   LIN {X -9.091, Y -16.998, Z 51.850} C_DIS
   LIN {X -7.957, Y -14.503, Z 51.850} C_DIS
   LIN {X -6.497, Y -10.839, Z 51.850} C_DIS
   LIN {X -6.440, Y -10.684, Z 51.850} C_DIS
   LIN {X -5.101, Y -6.672, Z 51.850} C_DIS
   LIN {X -4.128, Y -3.010, Z 51.850} C_DIS
   LIN {X -3.893, Y -2.128, Z 51.850} C_DIS
   LIN {X -3.542, Y -0.234, Z 51.850} C_DIS
   LIN {X -2.837, Y 3.485, Z 51.850} C_DIS
   LIN {X -2.656, Y 4.674, Z 51.850} C_DIS
   LIN {X -2.279, Y 9.653, Z 51.850} C_DIS
   LIN {X -2.115, Y 11.765, Z 51.850} C_DIS
   LIN {X -2.086, Y 12.130, Z 51.850} C_DIS
   LIN {X -2.030, Y 12.659, Z 51.850} C_DIS
   LIN {X -2.082, Y 13.927, Z 51.850} C_DIS
   LIN {X -2.664, Y 23.969, Z 51.850} C_DIS
   LIN {X -2.957, Y 25.919, Z 51.850} C_DIS
   LIN {X -3.415, Y 28.463, Z 51.850} C_DIS
   LIN {X -3.462, Y 28.724, Z 51.850} C_DIS
   LIN {X -3.657, Y 29.589, Z 51.850} C_DIS
   LIN {X -4.174, Y 31.893, Z 51.850} C_DIS
   LIN {X -4.435, Y 32.885, Z 51.850} C_DIS
   LIN {X -4.782, Y 34.185, Z 51.850} C_DIS
   LIN {X -5.293, Y 35.880, Z 51.850} C_DIS
   LIN {X -5.465, Y 36.456, Z 51.850} C_DIS
   LIN {X -5.565, Y 36.761, Z 51.850} C_DIS
   LIN {X -5.967, Y 37.975, Z 51.850} C_DIS
   LIN {X -6.308, Y 38.961, Z 51.850} C_DIS
   LIN {X -6.377, Y 39.157, Z 51.850} C_DIS
   LIN {X -6.424, Y 39.407, Z 51.850} C_DIS
   LIN {X -6.622, Y 40.453, Z 51.850} C_DIS
   LIN {X -6.434, Y 41.604, Z 51.850} C_DIS
   LIN {X -6.389, Y 41.872, Z 51.850} C_DIS
   LIN {X -6.240, Y 42.112, Z 51.850} C_DIS
   LIN {X -5.463, Y 43.327, Z 51.850} C_DIS
   LIN {X -3.784, Y 44.088, Z 51.850} C_DIS
   LIN {X -2.954, Y 44.485, Z 51.850} C_DIS
   LIN {X -2.346, Y 44.397, Z 51.850} C_DIS
   LIN {X -1.227, Y 44.232, Z 51.850}
   LaserEnd_Ext()
   LIN {X 8.602, Y 5.790, Z 51.850}
   LaserStart_Ext()
   LIN {X 8.602, Y -9.042, Z 51.850}
   LaserEnd_Ext()
   LIN {X 7.602, Y -17.948, Z 51.850}
   LaserStart_Ext()
   LIN {X 7.602, Y 15.368, Z 51.850}
   LaserEnd_Ext()
   LIN {X 6.602, Y 20.531, Z 51.850}
   LaserStart_Ext()
   LIN {X 6.602, Y -22.967, Z 51.850}
   LaserEnd_Ext()
   LIN {X 5.602, Y -25.282, Z 51.850}
   LaserStart_Ext()
   LIN {X 5.602, Y 25.306, Z 51.850}
   LaserEnd_Ext()
   LIN {X 4.602, Y 28.856, Z 51.850}
   LaserStart_Ext()
   LIN {X 4.602, Y -19.113, Z 51.850}
   LaserEnd_Ext()
   LIN {X 4.602, Y -22.901, Z 51.850}
   LaserStart_Ext()
   LIN {X 4.602, Y -26.434, Z 51.850}
   LaserEnd_Ext()
   LIN {X 3.602, Y -27.404, Z 51.850}
   LaserStart_Ext()
   LIN {X 3.602, Y -24.729, Z 51.850}
   LaserEnd_Ext()
   LIN {X 3.602, Y -17.421, Z 51.850}
   LaserStart_Ext()
   LIN {X 3.602, Y 32.251, Z 51.850}
   LaserEnd_Ext()
   LIN {X 2.602, Y 35.260, Z 51.850}
   LaserStart_Ext()
   LIN {X 2.602, Y -16.373, Z 51.850}
   LaserEnd_Ext()
   LIN {X 2.602, Y -25.693, Z 51.850}
   LaserStart_Ext()
   LIN {X 2.602, Y -27.986, Z 51.850}
   LaserEnd_Ext()
   LIN {X 1.602, Y -28.384, Z 51.850}
   LaserStart_Ext()
   LIN {X 1.602, Y -26.285, Z 51.850}
   LaserEnd_Ext()
   LIN {X 1.602, Y -15.740, Z 51.850}
   LaserStart_Ext()
   LIN {X 1.602, Y 37.974, Z 51.850}
   LaserEnd_Ext()
   LIN {X 0.602, Y 40.498, Z 51.850}
   LaserStart_Ext()
   LIN {X 0.602, Y -15.317, Z 51.850}
   LaserEnd_Ext()
   LIN {X 0.602, Y -26.624, Z 51.850}
   LaserStart_Ext()
   LIN {X 0.602, Y -28.775, Z 51.850}
   LaserEnd_Ext()
   LIN {X -0.398, Y -28.815, Z 51.850}
   LaserStart_Ext()
   LIN {X -0.398, Y -26.985, Z 51.850}
   LaserEnd_Ext()
   LIN {X -0.398, Y -15.189, Z 51.850}
   LaserStart_Ext()
   LIN {X -0.398, Y 42.404, Z 51.850}
   LaserEnd_Ext()
   LIN {X -1.398, Y 43.147, Z 51.850}
   LaserStart_Ext()
   LIN {X -1.398, Y 19.405, Z 51.850}
   LaserEnd_Ext()
   LIN {X -1.398, Y 8.047, Z 51.850}
   LaserStart_Ext()
   LIN {X -1.398, Y -15.067, Z 51.850}
   LaserEnd_Ext()
   LIN {X -1.398, Y -26.955, Z 51.850}
   LaserStart_Ext()
   LIN {X -1.398, Y -28.642, Z 51.850}
   LaserEnd_Ext()
   LIN {X -2.398, Y -28.469, Z 51.850}
   LaserStart_Ext()
   LIN {X -2.398, Y -26.818, Z 51.850}
   LaserEnd_Ext()
   LIN {X -2.398, Y -15.309, Z 51.850}
   LaserStart_Ext()
   LIN {X -2.398, Y 0.432, Z 51.850}
   LaserEnd_Ext()
   LIN {X -2.398, Y 28.460, Z 51.850}
   LaserStart_Ext()
   LIN {X -2.398, Y 43.394, Z 51.850}
   LaserEnd_Ext()
   LIN {X -3.398, Y 43.165, Z 51.850}
   LaserStart_Ext()
   LIN {X -3.398, Y 32.873, Z 51.850}
   LaserEnd_Ext()
   LIN {X -3.398, Y -4.158, Z 51.850}
   LaserStart_Ext()
   LIN {X -3.398, Y -15.630, Z 51.850}
   LaserEnd_Ext()
   LIN {X -3.398, Y -26.558, Z 51.850}
   LaserStart_Ext()
   LIN {X -3.398, Y -28.295, Z 51.850}
   LaserEnd_Ext()
   LIN {X -4.398, Y -28.122, Z 51.850}
   LaserStart_Ext()
   LIN {X -4.398, Y -25.932, Z 51.850}
   LaserEnd_Ext()
   LIN {X -4.398, Y -16.131, Z 51.850}
   LaserStart_Ext()
   LIN {X -4.398, Y -7.724, Z 51.850}
   LaserEnd_Ext()
   LIN {X -4.398, Y 36.378, Z 51.850}
   LaserStart_Ext()
   LIN {X -4.398, Y 42.712, Z 51.850}
   LaserEnd_Ext()
   LIN {X -5.398, Y 41.572, Z 51.850}
   LaserStart_Ext()
   LIN {X -5.398, Y 39.387, Z 51.850}
   LaserEnd_Ext()
   LIN {X -5.398, Y -10.720, Z 51.850}
   LaserStart_Ext()
   LIN {X -5.398, Y -17.051, Z 51.850}
   LaserEnd_Ext()
   LIN {X -5.398, Y -25.183, Z 51.850}
   LaserStart_Ext()
   LIN {X -5.398, Y -27.718, Z 51.850}
   LaserEnd_Ext()
   LIN {X -6.398, Y -26.934, Z 51.850}
   LaserStart_Ext()
   LIN {X -6.398, Y -23.699, Z 51.850}
   LaserEnd_Ext()
   LIN {X -6.398, Y -18.786, Z 51.850}
   LaserStart_Ext()
   LIN {X -6.398, Y -13.293, Z 51.850}
   LaserEnd_Ext()
   LIN {X -7.398, Y -15.691, Z 51.850}
   LaserStart_Ext()
   LIN {X -7.398, Y -25.741, Z 51.850}
   LaserEnd_Ext()
   LIN {X -8.398, Y -24.042, Z 51.850}
   LaserStart_Ext()
   LIN {X -8.398, Y -18.107, Z 51.850}
   LaserEnd_Ext()
   LIN {X 3.897, Y -22.048, Z 52.700}
   LaserStart_Ext()
   LIN {X 3.461, Y -23.044, Z 52.700} C_DIS
   LIN {X 3.108, Y -23.846, Z 52.700} C_DIS
   LIN {X 1.957, Y -24.884, Z 52.700} C_DIS
   LIN {X 1.508, Y -25.317, Z 52.700} C_DIS
   LIN {X 0.879, Y -25.530, Z 52.700} C_DIS
   LIN {X -0.660, Y -25.986, Z 52.700} C_DIS
   LIN {X -1.668, Y -25.850, Z 52.700} C_DIS
   LIN {X -2.710, Y -25.707, Z 52.700} C_DIS
   LIN {X -3.925, Y -24.947, Z 52.700} C_DIS
   LIN {X -4.462, Y -24.613, Z 52.700} C_DIS
   LIN {X -4.766, Y -24.167, Z 52.700} C_DIS
   LIN {X -5.630, Y -22.888, Z 52.700} C_DIS
   LIN {X -5.881, Y -21.409, Z 52.700} C_DIS
   LIN {X -5.980, Y -20.831, Z 52.700} C_DIS
   LIN {X -5.800, Y -20.305, Z 52.700} C_DIS
   LIN {X -5.042, Y -18.100, Z 52.700} C_DIS
   LIN {X -3.563, Y -16.747, Z 52.700} C_DIS
   LIN {X -3.489, Y -16.679, Z 52.700} C_DIS
   LIN {X -1.401, Y -16.013, Z 52.700} C_DIS
   LIN {X 0.253, Y -16.220, Z 52.700} C_DIS
   LIN {X 0.741, Y -16.280, Z 52.700} C_DIS
   LIN {X 1.229, Y -16.586, Z 52.700} C_DIS
   LIN {X 2.539, Y -17.413, Z 52.700} C_DIS
   LIN {X 3.482, Y -19.002, Z 52.700} C_DIS
   LIN {X 3.839, Y -19.599, Z 52.700} C_DIS
   LIN {X 3.868, Y -20.120, Z 52.700} C_DIS
   LIN {X 3.897, Y -22.048, Z 52.700}
   LaserEnd_Ext()
   LIN {X -6.440, Y 39.195, Z 52.700}
   LaserStart_Ext()
   LIN {X -6.031, Y 38.023, Z 52.700} C_DIS
   LIN {X -5.522, Y 36.495, Z 52.700} C_DIS
   LIN {X -5.003, Y 34.786, Z 52.700} C_DIS
   LIN {X -4.834, Y 34.226, Z 52.700} C_DIS
   LIN {X -4.622, Y 33.433, Z 52.700} C_DIS
   LIN {X -4.220, Y 31.936, Z 52.700} C_DIS
   LIN {X -4.160, Y 31.686, Z 52.700} C_DIS
   LIN {X -3.517, Y 28.844, Z 52.700} C_DIS
   LIN {X -3.238, Y 27.287, Z 52.700} C_DIS
   LIN {X -2.907, Y 25.444, Z 52.700} C_DIS
   LIN {X -2.694, Y 24.032, Z 52.700} C_DIS
   LIN {X -2.042, Y 12.765, Z 52.700} C_DIS
   LIN {X -2.035, Y 12.665, Z 52.700} C_DIS
   LIN {X -2.630, Y 4.802, Z 52.700} C_DIS
   LIN {X -2.918, Y 2.908, Z 52.700} C_DIS
   LIN {X -3.872, Y -2.129, Z 52.700} C_DIS
   LIN {X -3.961, Y -2.483, Z 52.700} C_DIS
   LIN {X -4.159, Y -3.222, Z 52.700} C_DIS
   LIN {X -5.120, Y -6.839, Z 52.700} C_DIS
   LIN {X -5.819, Y -8.933, Z 52.700} C_DIS
   LIN {X -6.431, Y -10.775, Z 52.700} C_DIS
   LIN {X -7.191, Y -12.703, Z 52.700} C_DIS
   LIN {X -7.896, Y -14.470, Z 52.700} C_DIS
   LIN {X -8.539, Y -15.886, Z 52.700} C_DIS
   LIN {X -9.111, Y -17.160, Z 52.700} C_DIS
   LIN {X -9.455, Y -18.416, Z 52.700} C_DIS
   LIN {X -9.956, Y -20.216, Z 52.700} C_DIS
   LIN {X -9.683, Y -22.635, Z 52.700} C_DIS
   LIN {X -9.534, Y -23.902, Z 52.700} C_DIS
   LIN {X -8.671, Y -25.359, Z 52.700} C_DIS
   LIN {X -7.628, Y -27.131, Z 52.700} C_DIS
   LIN {X -6.992, Y -27.631, Z 52.700} C_DIS
   LIN {X -5.335, Y -28.917, Z 52.700} C_DIS
   LIN {X -2.287, Y -29.446, Z 52.700} C_DIS
   LIN {X 0.367, Y -29.899, Z 52.700} C_DIS
   LIN {X 2.301, Y -29.198, Z 52.700} C_DIS
   LIN {X 3.776, Y -28.611, Z 52.700} C_DIS
   LIN {X 4.726, Y -27.690, Z 52.700} C_DIS
   LIN {X 6.373, Y -26.159, Z 52.700} C_DIS
   LIN {X 7.607, Y -23.279, Z 52.700} C_DIS
   LIN {X 7.870, Y -22.673, Z 52.700} C_DIS
   LIN {X 7.953, Y -22.225, Z 52.700} C_DIS
   LIN {X 8.447, Y -19.461, Z 52.700} C_DIS
   LIN {X 8.873, Y -16.648, Z 52.700} C_DIS
   LIN {X 8.891, Y -16.534, Z 52.700} C_DIS
   LIN {X 8.906, Y -16.414, Z 52.700} C_DIS
   LIN {X 9.346, Y -12.755, Z 52.700} C_DIS
   LIN {X 9.568, Y -10.105, Z 52.700} C_DIS
   LIN {X 9.732, Y -7.982, Z 52.700} C_DIS
   LIN {X 9.893, Y -2.443, Z 52.700} C_DIS
   LIN {X 9.924, Y -1.495, Z 52.700} C_DIS
   LIN {X 9.827, Y 1.258, Z 52.700} C_DIS
   LIN {X 9.794, Y 2.098, Z 52.700} C_DIS
   LIN {X 9.781, Y 4.353, Z 52.700} C_DIS
   LIN {X 9.137, Y 10.313, Z 52.700} C_DIS
   LIN {X 8.700, Y 14.833, Z 52.700} C_DIS
   LIN {X 7.579, Y 20.715, Z 52.700} C_DIS
   LIN {X 6.563, Y 25.567, Z 52.700} C_DIS
   LIN {X 5.392, Y 29.673, Z 52.700} C_DIS
   LIN {X 4.526, Y 32.613, Z 52.700} C_DIS
   LIN {X 4.051, Y 34.041, Z 52.700} C_DIS
   LIN {X 3.564, Y 35.455, Z 52.700} C_DIS
   LIN {X 3.153, Y 36.583, Z 52.700} C_DIS
   LIN {X 2.877, Y 37.340, Z 52.700} C_DIS
   LIN {X 2.446, Y 38.454, Z 52.700} C_DIS
   LIN {X 2.118, Y 39.311, Z 52.700} C_DIS
   LIN {X 1.886, Y 39.889, Z 52.700} C_DIS
   LIN {X 1.543, Y 40.733, Z 52.700} C_DIS
   LIN {X 1.075, Y 41.846, Z 52.700} C_DIS
   LIN {X 0.968, Y 42.102, Z 52.700} C_DIS
   LIN {X 0.846, Y 42.287, Z 52.700} C_DIS
   LIN {X 0.152, Y 43.327, Z 52.700} C_DIS
   LIN {X -1.096, Y 44.147, Z 52.700} C_DIS
   LIN {X -1.303, Y 44.282, Z 52.700} C_DIS
   LIN {X -1.744, Y 44.345, Z 52.700} C_DIS
   LIN {X -3.030, Y 44.531, Z 52.700} C_DIS
   LIN {X -5.347, Y 43.424, Z 52.700} C_DIS
   LIN {X -5.565, Y 43.330, Z 52.700} C_DIS
   LIN {X -5.657, Y 43.211, Z 52.700} C_DIS
   LIN {X -6.452, Y 41.928, Z 52.700} C_DIS
   LIN {X -6.652, Y 40.735, Z 52.700} C_DIS
   LIN {X -6.689, Y 40.519, Z 52.700} C_DIS
   LIN {X -6.649, Y 40.300, Z 52.700} C_DIS
   LIN {X -6.440, Y 39.195, Z 52.700}
   LaserEnd_Ext()
   LIN {X -0.513, Y 42.522, Z 52.700}
   LaserStart_Ext()
   LIN {X -4.907, Y 42.522, Z 52.700}
   LaserEnd_Ext()
   LIN {X -5.506, Y 41.522, Z 52.700}
   LaserStart_Ext()
   LIN {X 0.127, Y 41.522, Z 52.700}
   LaserEnd_Ext()
   LIN {X 0.547, Y 40.522, Z 52.700}
   LaserStart_Ext()
   LIN {X -5.673, Y 40.522, Z 52.700}
   LaserEnd_Ext()
   LIN {X -5.484, Y 39.522, Z 52.700}
   LaserStart_Ext()
   LIN {X 0.956, Y 39.522, Z 52.700}
   LaserEnd_Ext()
   LIN {X 1.350, Y 38.522, Z 52.700}
   LaserStart_Ext()
   LIN {X -5.146, Y 38.522, Z 52.700}
   LaserEnd_Ext()
   LIN {X -4.810, Y 37.522, Z 52.700}
   LaserStart_Ext()
   LIN {X 1.735, Y 37.522, Z 52.700}
   LaserEnd_Ext()
   LIN {X 2.111, Y 36.522, Z 52.700}
   LaserStart_Ext()
   LIN {X -4.485, Y 36.522, Z 52.700}
   LaserEnd_Ext()
   LIN {X -4.181, Y 35.522, Z 52.700}
   LaserStart_Ext()
   LIN {X 2.475, Y 35.522, Z 52.700}
   LaserEnd_Ext()
   LIN {X 2.828, Y 34.522, Z 52.700}
   LaserStart_Ext()
   LIN {X -3.879, Y 34.522, Z 52.700}
   LaserEnd_Ext()
   LIN {X -3.611, Y 33.522, Z 52.700}
   LaserStart_Ext()
   LIN {X 3.170, Y 33.522, Z 52.700}
   LaserEnd_Ext()
   LIN {X 3.503, Y 32.522, Z 52.700}
   LaserStart_Ext()
   LIN {X -3.342, Y 32.522, Z 52.700}
   LaserEnd_Ext()
   LIN {X -3.097, Y 31.522, Z 52.700}
   LaserStart_Ext()
   LIN {X 3.805, Y 31.522, Z 52.700}
   LaserEnd_Ext()
   LIN {X 4.100, Y 30.522, Z 52.700}
   LaserStart_Ext()
   LIN {X -2.871, Y 30.522, Z 52.700}
   LaserEnd_Ext()
   LIN {X -2.645, Y 29.522, Z 52.700}
   LaserStart_Ext()
   LIN {X 4.394, Y 29.522, Z 52.700}
   LaserEnd_Ext()
   LIN {X 4.681, Y 28.522, Z 52.700}
   LaserStart_Ext()
   LIN {X -2.443, Y 28.522, Z 52.700}
   LaserEnd_Ext()
   LIN {X -2.264, Y 27.522, Z 52.700}
   LaserStart_Ext()
   LIN {X 4.966, Y 27.522, Z 52.700}
   LaserEnd_Ext()
   LIN {X 5.251, Y 26.522, Z 52.700}
   LaserStart_Ext()
   LIN {X -2.084, Y 26.522, Z 52.700}
   LaserEnd_Ext()
   LIN {X -1.907, Y 25.522, Z 52.700}
   LaserStart_Ext()
   LIN {X 5.536, Y 25.522, Z 52.700}
   LaserEnd_Ext()
   LIN {X 5.760, Y 24.522, Z 52.700}
   LaserStart_Ext()
   LIN {X -1.757, Y 24.522, Z 52.700}
   LaserEnd_Ext()
   LIN {X -1.663, Y 23.522, Z 52.700}
   LaserStart_Ext()
   LIN {X 5.969, Y 23.522, Z 52.700}
   LaserEnd_Ext()
   LIN {X 6.179, Y 22.522, Z 52.700}
   LaserStart_Ext()
   LIN {X -1.605, Y 22.522, Z 52.700}
   LaserEnd_Ext()
   LIN {X -1.547, Y 21.522, Z 52.700}
   LaserStart_Ext()
   LIN {X 6.388, Y 21.522, Z 52.700}
   LaserEnd_Ext()
   LIN {X 6.598, Y 20.522, Z 52.700}
   LaserStart_Ext()
   LIN {X -1.489, Y 20.522, Z 52.700}
   LaserEnd_Ext()
   LIN {X -1.431, Y 19.522, Z 52.700}
   LaserStart_Ext()
   LIN {X 6.788, Y 19.522, Z 52.700}
   LaserEnd_Ext()
   LIN {X 6.979, Y 18.522, Z 52.700}
   LaserStart_Ext()
   LIN {X -1.373, Y 18.522, Z 52.700}
   LaserEnd_Ext()
   LIN {X -1.316, Y 17.522, Z 52.700}
   LaserStart_Ext()
   LIN {X 7.169, Y 17.522, Z 52.700}
   LaserEnd_Ext()
   LIN {X 7.360, Y 16.522, Z 52.700}
   LaserStart_Ext()
   LIN {X -1.258, Y 16.522, Z 52.700}
   LaserEnd_Ext()
   LIN {X -1.200, Y 15.522, Z 52.700}
   LaserStart_Ext()
   LIN {X 7.550, Y 15.522, Z 52.700}
   LaserEnd_Ext()
   LIN {X 7.725, Y 14.522, Z 52.700}
   LaserStart_Ext()
   LIN {X -1.142, Y 14.522, Z 52.700}
   LaserEnd_Ext()
   LIN {X -1.084, Y 13.522, Z 52.700}
   LaserStart_Ext()
   LIN {X 7.822, Y 13.522, Z 52.700}
   LaserEnd_Ext()
   LIN {X 7.919, Y 12.522, Z 52.700}
   LaserStart_Ext()
   LIN {X -1.042, Y 12.522, Z 52.700}
   LaserEnd_Ext()
   LIN {X -1.118, Y 11.522, Z 52.700}
   LaserStart_Ext()
   LIN {X 8.015, Y 11.522, Z 52.700}
   LaserEnd_Ext()
   LIN {X 8.112, Y 10.522, Z 52.700}
   LaserStart_Ext()
   LIN {X -1.194, Y 10.522, Z 52.700}
   LaserEnd_Ext()
   LIN {X -1.269, Y 9.522, Z 52.700}
   LaserStart_Ext()
   LIN {X 8.216, Y 9.522, Z 52.700}
   LaserEnd_Ext()
   LIN {X 8.324, Y 8.522, Z 52.700}
   LaserStart_Ext()
   LIN {X -1.345, Y 8.522, Z 52.700}
   LaserEnd_Ext()
   LIN {X -1.421, Y 7.522, Z 52.700}
   LaserStart_Ext()
   LIN {X 8.433, Y 7.522, Z 52.700}
   LaserEnd_Ext()
   LIN {X 8.541, Y 6.522, Z 52.700}
   LaserStart_Ext()
   LIN {X -1.497, Y 6.522, Z 52.700}
   LaserEnd_Ext()
   LIN {X -1.572, Y 5.522, Z 52.700}
   LaserStart_Ext()
   LIN {X 8.649, Y 5.522, Z 52.700}
   LaserEnd_Ext()
   LIN {X 8.757, Y 4.522, Z 52.700}
   LaserStart_Ext()
   LIN {X -1.661, Y 4.522, Z 52.700}
   LaserEnd_Ext()
   LIN {X -1.813, Y 3.522, Z 52.700}
   LaserStart_Ext()
   LIN {X 8.786, Y 3.522, Z 52.700}
   LaserEnd_Ext()
   LIN {X 8.791, Y 2.522, Z 52.700}
   LaserStart_Ext()
   LIN {X -1.974, Y 2.522, Z 52.700}
   LaserEnd_Ext()
   LIN {X -2.163, Y 1.522, Z 52.700}
   LaserStart_Ext()
   LIN {X 8.816, Y 1.522, Z 52.700}
   LaserEnd_Ext()
   LIN {X 8.852, Y 0.522, Z 52.700}
   LaserStart_Ext()
   LIN {X -2.352, Y 0.522, Z 52.700}
   LaserEnd_Ext()
   LIN {X -2.542, Y -0.478, Z 52.700}
   LaserStart_Ext()
   LIN {X 8.888, Y -0.478, Z 52.700}
   LaserEnd_Ext()
   LIN {X 8.923, Y -1.478, Z 52.700}
   LaserStart_Ext()
   LIN {X -2.731, Y -1.478, Z 52.700}
   LaserEnd_Ext()
   LIN {X -2.929, Y -2.478, Z 52.700}
   LaserStart_Ext()
   LIN {X 8.891, Y -2.478, Z 52.700}
   LaserEnd_Ext()
   LIN {X 8.862, Y -3.478, Z 52.700}
   LaserStart_Ext()
   LIN {X -3.192, Y -3.478, Z 52.700}
   LaserEnd_Ext()
   LIN {X -3.458, Y -4.478, Z 52.700}
   LaserStart_Ext()
   LIN {X 8.833, Y -4.478, Z 52.700}
   LaserEnd_Ext()
   LIN {X 8.804, Y -5.478, Z 52.700}
   LaserStart_Ext()
   LIN {X -3.724, Y -5.478, Z 52.700}
   LaserEnd_Ext()
   LIN {X -3.990, Y -6.478, Z 52.700}
   LaserStart_Ext()
   LIN {X 8.775, Y -6.478, Z 52.700}
   LaserEnd_Ext()
   LIN {X 8.746, Y -7.478, Z 52.700}
   LaserStart_Ext()
   LIN {X -4.279, Y -7.478, Z 52.700}
   LaserEnd_Ext()
   LIN {X -4.613, Y -8.478, Z 52.700}
   LaserStart_Ext()
   LIN {X 8.691, Y -8.478, Z 52.700}
   LaserEnd_Ext()
   LIN {X 8.614, Y -9.478, Z 52.700}
   LaserStart_Ext()
   LIN {X -4.947, Y -9.478, Z 52.700}
   LaserEnd_Ext()
   LIN {X -5.279, Y -10.478, Z 52.700}
   LaserStart_Ext()
   LIN {X 8.533, Y -10.478, Z 52.700}
   LaserEnd_Ext()
   LIN {X 8.449, Y -11.478, Z 52.700}
   LaserStart_Ext()
   LIN {X -5.633, Y -11.478, Z 52.700}
   LaserEnd_Ext()
   LIN {X -6.028, Y -12.478, Z 52.700}
   LaserStart_Ext()
   LIN {X 8.365, Y -12.478, Z 52.700}
   LaserEnd_Ext()
   LIN {X 8.252, Y -13.478, Z 52.700}
   LaserStart_Ext()
   LIN {X -6.424, Y -13.478, Z 52.700}
   LaserEnd_Ext()
   LIN {X -6.822, Y -14.478, Z 52.700}
   LaserStart_Ext()
   LIN {X 8.131, Y -14.478, Z 52.700}
   LaserEnd_Ext()
   LIN {X 8.011, Y -15.478, Z 52.700}
   LaserStart_Ext()
   LIN {X 1.345, Y -15.478, Z 52.700}
   LaserEnd_Ext()
   LIN {X -3.016, Y -15.478, Z 52.700}
   LaserStart_Ext()
   LIN {X -7.255, Y -15.478, Z 52.700}
   LaserEnd_Ext()
   LIN {X -7.709, Y -16.478, Z 52.700}
   LaserStart_Ext()
   LIN {X -4.751, Y -16.478, Z 52.700}
   LaserEnd_Ext()
   LIN {X 2.932, Y -16.478, Z 52.700}
   LaserStart_Ext()
   LIN {X 7.887, Y -16.478, Z 52.700}
   LaserEnd_Ext()
   LIN {X 7.736, Y -17.478, Z 52.700}
   LaserStart_Ext()
   LIN {X 3.740, Y -17.478, Z 52.700}
   LaserEnd_Ext()
   LIN {X -5.824, Y -17.478, Z 52.700}
   LaserStart_Ext()
   LIN {X -8.158, Y -17.478, Z 52.700}
   LaserEnd_Ext()
   LIN {X -8.435, Y -18.478, Z 52.700}
   LaserStart_Ext()
   LIN {X -6.229, Y -18.478, Z 52.700}
   LaserEnd_Ext()
   LIN {X 4.334, Y -18.478, Z 52.700}
   LaserStart_Ext()
   LIN {X 7.585, Y -18.478, Z 52.700}
   LaserEnd_Ext()
   LIN {X 7.428, Y -19.478, Z 52.700}
   LaserStart_Ext()
   LIN {X 4.830, Y -19.478, Z 52.700}
   LaserEnd_Ext()
   LIN {X -6.573, Y -19.478, Z 52.700}
   LaserStart_Ext()
   LIN {X -8.713, Y -19.478, Z 52.700}
   LaserEnd_Ext()
   LIN {X -8.920, Y -20.478, Z 52.700}
   LaserStart_Ext()
   LIN {X -6.916, Y -20.478, Z 52.700}
   LaserEnd_Ext()
   LIN {X 4.873, Y -20.478, Z 52.700}
   LaserStart_Ext()
   LIN {X 7.250, Y -20.478, Z 52.700}
   LaserEnd_Ext()
   LIN {X 7.071, Y -21.478, Z 52.700}
   LaserStart_Ext()
   LIN {X 4.889, Y -21.478, Z 52.700}
   LaserEnd_Ext()
   LIN {X -6.883, Y -21.478, Z 52.700}
   LaserStart_Ext()
   LIN {X -8.808, Y -21.478, Z 52.700}
   LaserEnd_Ext()
   LIN {X -8.695, Y -22.478, Z 52.700}
   LaserStart_Ext()
   LIN {X -6.714, Y -22.478, Z 52.700}
   LaserEnd_Ext()
   LIN {X 4.801, Y -22.478, Z 52.700}
   LaserStart_Ext()
   LIN {X 6.865, Y -22.478, Z 52.700}
   LaserEnd_Ext()
   LIN {X 6.434, Y -23.478, Z 52.700}
   LaserStart_Ext()
   LIN {X 4.362, Y -23.478, Z 52.700}
   LaserEnd_Ext()
   LIN {X -6.438, Y -23.478, Z 52.700}
   LaserStart_Ext()
   LIN {X -8.577, Y -23.478, Z 52.700}
   LaserEnd_Ext()
   LIN {X -8.031, Y -24.478, Z 52.700}
   LaserStart_Ext()
   LIN {X -5.762, Y -24.478, Z 52.700}
   LaserEnd_Ext()
   LIN {X 3.881, Y -24.478, Z 52.700}
   LaserStart_Ext()
   LIN {X 6.006, Y -24.478, Z 52.700}
   LaserEnd_Ext()
   LIN {X 5.577, Y -25.478, Z 52.700}
   LaserStart_Ext()
   LIN {X 2.791, Y -25.478, Z 52.700}
   LaserEnd_Ext()
   LIN {X -4.964, Y -25.478, Z 52.700}
   LaserStart_Ext()
   LIN {X -7.441, Y -25.478, Z 52.700}
   LaserEnd_Ext()
   LIN {X -6.840, Y -26.478, Z 52.700}
   LaserStart_Ext()
   LIN {X -3.363, Y -26.478, Z 52.700}
   LaserEnd_Ext()
   LIN {X 1.195, Y -26.478, Z 52.700}
   LaserStart_Ext()
   LIN {X 4.560, Y -26.478, Z 52.700}
   LaserEnd_Ext()
   LIN {X 3.507, Y -27.478, Z 52.700}
   LaserStart_Ext()
   LIN {X -5.558, Y -27.478, Z 52.700}
   LaserEnd_Ext()
   LIN {X -2.010, Y -28.478, Z 52.700}
   LaserStart_Ext()
   LIN {X 1.352, Y -28.478, Z 52.700}
   LaserEnd_Ext()
   LIN {X -2.322, Y -25.700, Z 53.550}
   LaserStart_Ext()
   LIN {X -2.621, Y -25.660, Z 53.550} C_DIS
   LIN {X -2.815, Y -25.541, Z 53.550} C_DIS
   LIN {X -4.376, Y -24.570, Z 53.550} C_DIS
   LIN {X -5.507, Y -22.909, Z 53.550} C_DIS
   LIN {X -5.560, Y -22.779, Z 53.550} C_DIS
   LIN {X -5.903, Y -20.792, Z 53.550} C_DIS
   LIN {X -5.283, Y -18.984, Z 53.550} C_DIS
   LIN {X -4.960, Y -18.043, Z 53.550} C_DIS
   LIN {X -3.418, Y -16.632, Z 53.550} C_DIS
   LIN {X -1.805, Y -16.113, Z 53.550} C_DIS
   LIN {X -1.333, Y -15.963, Z 53.550} C_DIS
   LIN {X -0.975, Y -16.008, Z 53.550} C_DIS
   LIN {X 0.808, Y -16.225, Z 53.550} C_DIS
   LIN {X 2.587, Y -17.340, Z 53.550} C_DIS
   LIN {X 3.913, Y -19.536, Z 53.550} C_DIS
   LIN {X 4.018, Y -21.420, Z 53.550} C_DIS
   LIN {X 4.024, Y -21.790, Z 53.550} C_DIS
   LIN {X 3.940, Y -21.981, Z 53.550} C_DIS
   LIN {X 3.082, Y -23.933, Z 53.550} C_DIS
   LIN {X 1.954, Y -24.949, Z 53.550} C_DIS
   LIN {X 1.520, Y -25.311, Z 53.550} C_DIS
   LIN {X 0.629, Y -25.576, Z 53.550} C_DIS
   LIN {X -0.583, Y -25.935, Z 53.550} C_DIS
   LIN {X -2.322, Y -25.700, Z 53.550}
   LaserEnd_Ext()
   LIN {X -1.378, Y 44.332, Z 53.550}
   LaserStart_Ext()
   LIN {X -2.427, Y 44.482, Z 53.550} C_DIS
   LIN {X -3.106, Y 44.576, Z 53.550} C_DIS
   LIN {X -3.989, Y 44.311, Z 53.550} C_DIS
   LIN {X -4.992, Y 43.880, Z 53.550} C_DIS
   LIN {X -5.741, Y 43.267, Z 53.550} C_DIS
   LIN {X -6.331, Y 42.297, Z 53.550} C_DIS
   LIN {X -6.511, Y 41.995, Z 53.550} C_DIS
   LIN {X -6.587, Y 41.589, Z 53.550} C_DIS
   LIN {X -6.756, Y 40.620, Z 53.550} C_DIS
   LIN {X -6.582, Y 39.670, Z 53.550} C_DIS
   LIN {X -6.504, Y 39.233, Z 53.550} C_DIS
   LIN {X -6.415, Y 38.981, Z 53.550} C_DIS
   LIN {X -6.089, Y 38.052, Z 53.550} C_DIS
   LIN {X -5.656, Y 36.766, Z 53.550} C_DIS
   LIN {X -5.579, Y 36.535, Z 53.550} C_DIS
   LIN {X -5.448, Y 36.102, Z 53.550} C_DIS
   LIN {X -4.886, Y 34.268, Z 53.550} C_DIS
   LIN {X -4.504, Y 32.861, Z 53.550} C_DIS
   LIN {X -4.267, Y 31.979, Z 53.550} C_DIS
   LIN {X -4.078, Y 31.199, Z 53.550} C_DIS
   LIN {X -3.572, Y 28.963, Z 53.550} C_DIS
   LIN {X -3.061, Y 26.110, Z 53.550} C_DIS
   LIN {X -2.856, Y 24.970, Z 53.550} C_DIS
   LIN {X -2.725, Y 24.096, Z 53.550} C_DIS
   LIN {X -2.321, Y 17.122, Z 53.550} C_DIS
   LIN {X -2.118, Y 13.905, Z 53.550} C_DIS
   LIN {X -2.037, Y 12.794, Z 53.550} C_DIS
   LIN {X -2.086, Y 11.765, Z 53.550} C_DIS
   LIN {X -2.603, Y 4.930, Z 53.550} C_DIS
   LIN {X -2.999, Y 2.331, Z 53.550} C_DIS
   LIN {X -3.800, Y -1.898, Z 53.550} C_DIS
   LIN {X -4.187, Y -3.451, Z 53.550} C_DIS
   LIN {X -5.059, Y -6.703, Z 53.550} C_DIS
   LIN {X -5.139, Y -7.006, Z 53.550} C_DIS
   LIN {X -5.198, Y -7.182, Z 53.550} C_DIS
   LIN {X -6.397, Y -10.791, Z 53.550} C_DIS
   LIN {X -7.777, Y -14.292, Z 53.550} C_DIS
   LIN {X -7.834, Y -14.438, Z 53.550} C_DIS
   LIN {X -9.043, Y -17.128, Z 53.550} C_DIS
   LIN {X -9.796, Y -19.882, Z 53.550} C_DIS
   LIN {X -9.881, Y -20.186, Z 53.550} C_DIS
   LIN {X -9.835, Y -20.595, Z 53.550} C_DIS
   LIN {X -9.450, Y -23.871, Z 53.550} C_DIS
   LIN {X -7.709, Y -26.809, Z 53.550} C_DIS
   LIN {X -7.536, Y -27.096, Z 53.550} C_DIS
   LIN {X -7.107, Y -27.427, Z 53.550} C_DIS
   LIN {X -5.239, Y -28.876, Z 53.550} C_DIS
   LIN {X -3.702, Y -29.143, Z 53.550} C_DIS
   LIN {X 0.435, Y -29.849, Z 53.550} C_DIS
   LIN {X 3.449, Y -28.758, Z 53.550} C_DIS
   LIN {X 3.716, Y -28.651, Z 53.550} C_DIS
   LIN {X 3.888, Y -28.485, Z 53.550} C_DIS
   LIN {X 6.460, Y -26.095, Z 53.550} C_DIS
   LIN {X 7.627, Y -23.372, Z 53.550} C_DIS
   LIN {X 7.952, Y -22.601, Z 53.550} C_DIS
   LIN {X 8.119, Y -21.640, Z 53.550} C_DIS
   LIN {X 8.522, Y -19.388, Z 53.550} C_DIS
   LIN {X 8.795, Y -17.581, Z 53.550} C_DIS
   LIN {X 8.958, Y -16.459, Z 53.550} C_DIS
   LIN {X 9.220, Y -14.215, Z 53.550} C_DIS
   LIN {X 9.404, Y -12.679, Z 53.550} C_DIS
   LIN {X 9.489, Y -11.665, Z 53.550} C_DIS
   LIN {X 9.779, Y -7.905, Z 53.550} C_DIS
   LIN {X 9.918, Y -3.112, Z 53.550} C_DIS
   LIN {X 9.956, Y -1.393, Z 53.550} C_DIS
   LIN {X 9.914, Y -0.089, Z 53.550} C_DIS
   LIN {X 9.836, Y 2.115, Z 53.550} C_DIS
   LIN {X 9.813, Y 2.710, Z 53.550} C_DIS
   LIN {X 9.803, Y 4.306, Z 53.550} C_DIS
   LIN {X 9.348, Y 8.526, Z 53.550} C_DIS
   LIN {X 8.800, Y 14.191, Z 53.550} C_DIS
   LIN {X 7.394, Y 21.566, Z 53.550} C_DIS
   LIN {X 6.595, Y 25.385, Z 53.550} C_DIS
   LIN {X 5.117, Y 30.569, Z 53.550} C_DIS
   LIN {X 4.676, Y 32.064, Z 53.550} C_DIS
   LIN {X 3.903, Y 34.387, Z 53.550} C_DIS
   LIN {X 3.697, Y 34.986, Z 53.550} C_DIS
   LIN {X 3.523, Y 35.464, Z 53.550} C_DIS
   LIN {X 2.780, Y 37.502, Z 53.550} C_DIS
   LIN {X 2.465, Y 38.316, Z 53.550} C_DIS
   LIN {X 2.058, Y 39.361, Z 53.550} C_DIS
   LIN {X 1.678, Y 40.291, Z 53.550} C_DIS
   LIN {X 1.476, Y 40.790, Z 53.550} C_DIS
   LIN {X 1.320, Y 41.162, Z 53.550} C_DIS
   LIN {X 0.898, Y 42.157, Z 53.550} C_DIS
   LIN {X 0.111, Y 43.332, Z 53.550} C_DIS
   LIN {X 0.038, Y 43.407, Z 53.550} C_DIS
   LIN {X -1.378, Y 44.332, Z 53.550}
   LaserEnd_Ext()
   LIN {X -8.280, Y -18.129, Z 53.550}
   LaserStart_Ext()
   LIN {X -8.280, Y -23.884, Z 53.550}
   LaserEnd_Ext()
   LIN {X -7.280, Y -25.572, Z 53.550}
   LaserStart_Ext()
   LIN {X -7.280, Y -15.645, Z 53.550}
   LaserEnd_Ext()
   LIN {X -6.280, Y -13.220, Z 53.550}
   LaserStart_Ext()
   LIN {X -6.280, Y -18.807, Z 53.550}
   LaserEnd_Ext()
   LIN {X -6.280, Y -23.551, Z 53.550}
   LaserStart_Ext()
   LIN {X -6.280, Y -26.803, Z 53.550}
   LaserEnd_Ext()
   LIN {X -5.280, Y -27.579, Z 53.550}
   LaserStart_Ext()
   LIN {X -5.280, Y -25.019, Z 53.550}
   LaserEnd_Ext()
   LIN {X -5.280, Y -16.981, Z 53.550}
   LaserStart_Ext()
   LIN {X -5.280, Y -10.601, Z 53.550}
   LaserEnd_Ext()
   LIN {X -5.280, Y 38.768, Z 53.550}
   LaserStart_Ext()
   LIN {X -5.280, Y 42.100, Z 53.550}
   LaserEnd_Ext()
   LIN {X -4.280, Y 43.097, Z 53.550}
   LaserStart_Ext()
   LIN {X -4.280, Y 35.704, Z 53.550}
   LaserEnd_Ext()
   LIN {X -4.280, Y -7.590, Z 53.550}
   LaserStart_Ext()
   LIN {X -4.280, Y -16.065, Z 53.550}
   LaserEnd_Ext()
   LIN {X -4.280, Y -25.807, Z 53.550}
   LaserStart_Ext()
   LIN {X -4.280, Y -28.028, Z 53.550}
   LaserEnd_Ext()
   LIN {X -3.280, Y -28.201, Z 53.550}
   LaserStart_Ext()
   LIN {X -3.280, Y -26.429, Z 53.550}
   LaserEnd_Ext()
   LIN {X -3.280, Y -15.537, Z 53.550}
   LaserStart_Ext()
   LIN {X -3.280, Y -3.928, Z 53.550}
   LaserEnd_Ext()
   LIN {X -3.280, Y 32.152, Z 53.550}
   LaserStart_Ext()
   LIN {X -3.280, Y 43.480, Z 53.550}
   LaserEnd_Ext()
   LIN {X -2.280, Y 43.451, Z 53.550}
   LaserStart_Ext()
   LIN {X -2.280, Y 27.420, Z 53.550}
   LaserEnd_Ext()
   LIN {X -2.280, Y 0.754, Z 53.550}
   LaserStart_Ext()
   LIN {X -2.280, Y -15.216, Z 53.550}
   LaserEnd_Ext()
   LIN {X -2.280, Y -26.715, Z 53.550}
   LaserStart_Ext()
   LIN {X -2.280, Y -28.371, Z 53.550}
   LaserEnd_Ext()
   LIN {X -1.280, Y -28.542, Z 53.550}
   LaserStart_Ext()
   LIN {X -1.280, Y -26.850, Z 53.550}
   LaserEnd_Ext()
   LIN {X -1.280, Y -14.965, Z 53.550}
   LaserStart_Ext()
   LIN {X -1.280, Y 9.162, Z 53.550}
   LaserEnd_Ext()
   LIN {X -1.280, Y 16.504, Z 53.550}
   LaserStart_Ext()
   LIN {X -1.280, Y 43.073, Z 53.550}
   LaserEnd_Ext()
   LIN {X -0.280, Y 42.118, Z 53.550}
   LaserStart_Ext()
   LIN {X -0.280, Y -15.085, Z 53.550}
   LaserEnd_Ext()
   LIN {X -0.280, Y -26.888, Z 53.550}
   LaserStart_Ext()
   LIN {X -0.280, Y -28.713, Z 53.550}
   LaserEnd_Ext()
   LIN {X 0.720, Y -28.682, Z 53.550}
   LaserStart_Ext()
   LIN {X 0.720, Y -26.592, Z 53.550}
   LaserEnd_Ext()
   LIN {X 0.720, Y -15.207, Z 53.550}
   LaserStart_Ext()
   LIN {X 0.720, Y 39.993, Z 53.550}
   LaserEnd_Ext()
   LIN {X 1.720, Y 37.469, Z 53.550}
   LaserStart_Ext()
   LIN {X 1.720, Y -15.617, Z 53.550}
   LaserEnd_Ext()
   LIN {X 1.720, Y -26.295, Z 53.550}
   LaserStart_Ext()
   LIN {X 1.720, Y -28.320, Z 53.550}
   LaserEnd_Ext()
   LIN {X 2.720, Y -27.958, Z 53.550}
   LaserStart_Ext()
   LIN {X 2.720, Y -25.605, Z 53.550}
   LaserEnd_Ext()
   LIN {X 2.720, Y -16.244, Z 53.550}
   LaserStart_Ext()
   LIN {X 2.720, Y 34.745, Z 53.550}
   LaserEnd_Ext()
   LIN {X 3.720, Y 31.771, Z 53.550}
   LaserStart_Ext()
   LIN {X 3.720, Y -17.265, Z 53.550}
   LaserEnd_Ext()
   LIN {X 3.720, Y -24.704, Z 53.550}
   LaserStart_Ext()
   LIN {X 3.720, Y -27.276, Z 53.550}
   LaserEnd_Ext()
   LIN {X 4.720, Y -26.347, Z 53.550}
   LaserStart_Ext()
   LIN {X 4.720, Y -22.691, Z 53.550}
   LaserEnd_Ext()
   LIN {X 4.720, Y -18.938, Z 53.550}
   LaserStart_Ext()
   LIN {X 4.720, Y 28.313, Z 53.550}
   LaserEnd_Ext()
   LIN {X 5.720, Y 24.682, Z 53.550}
   LaserStart_Ext()
   LIN {X 5.720, Y -25.283, Z 53.550}
   LaserEnd_Ext()
   LIN {X 6.720, Y -22.949, Z 53.550}
   LaserStart_Ext()
   LIN {X 6.720, Y 19.762, Z 53.550}
   LaserEnd_Ext()
   LIN {X 7.720, Y 14.514, Z 53.550}
   LaserStart_Ext()
   LIN {X 7.720, Y -18.001, Z 53.550}
   LaserEnd_Ext()
   LIN {X 8.720, Y -8.631, Z 53.550}
   LaserStart_Ext()
   LIN {X 8.720, Y 5.023, Z 53.550}
   LaserEnd_Ext()
   LIN {X -3.891, Y -24.775, Z 54.400}
   LaserStart_Ext()
   LIN {X -4.289, Y -24.527, Z 54.400} C_DIS
   LIN {X -4.600, Y -24.071, Z 54.400} C_DIS
   LIN {X -5.466, Y -22.808, Z 54.400} C_DIS
   LIN {X -5.715, Y -21.394, Z 54.400} C_DIS
   LIN {X -5.826, Y -20.753, Z 54.400} C_DIS
   LIN {X -5.232, Y -19.021, Z 54.400} C_DIS
   LIN {X -4.880, Y -17.989, Z 54.400} C_DIS
   LIN {X -4.574, Y -17.708, Z 54.400} C_DIS
   LIN {X -3.349, Y -16.586, Z 54.400} C_DIS
   LIN {X -2.128, Y -16.193, Z 54.400} C_DIS
   LIN {X -1.262, Y -15.912, Z 54.400} C_DIS
   LIN {X -0.085, Y -16.053, Z 54.400} C_DIS
   LIN {X 0.875, Y -16.170, Z 54.400} C_DIS
   LIN {X 1.549, Y -16.592, Z 54.400} C_DIS
   LIN {X 2.677, Y -17.294, Z 54.400} C_DIS
   LIN {X 3.503, Y -18.664, Z 54.400} C_DIS
   LIN {X 3.988, Y -19.474, Z 54.400} C_DIS
   LIN {X 4.041, Y -20.428, Z 54.400} C_DIS
   LIN {X 4.115, Y -21.681, Z 54.400} C_DIS
   LIN {X 3.861, Y -22.276, Z 54.400} C_DIS
   LIN {X 3.468, Y -23.082, Z 54.400} C_DIS
   LIN {X 3.056, Y -24.019, Z 54.400} C_DIS
   LIN {X 2.653, Y -24.382, Z 54.400} C_DIS
   LIN {X 1.603, Y -25.257, Z 54.400} C_DIS
   LIN {X -0.431, Y -25.862, Z 54.400} C_DIS
   LIN {X -0.553, Y -25.878, Z 54.400} C_DIS
   LIN {X -2.532, Y -25.613, Z 54.400} C_DIS
   LIN {X -3.891, Y -24.775, Z 54.400}
   LaserEnd_Ext()
   LIN {X -1.453, Y 44.382, Z 54.400}
   LaserStart_Ext()
   LIN {X -1.910, Y 44.444, Z 54.400} C_DIS
   LIN {X -3.182, Y 44.622, Z 54.400} C_DIS
   LIN {X -4.016, Y 44.371, Z 54.400} C_DIS
   LIN {X -5.081, Y 43.903, Z 54.400} C_DIS
   LIN {X -5.847, Y 43.269, Z 54.400} C_DIS
   LIN {X -6.117, Y 42.829, Z 54.400} C_DIS
   LIN {X -6.558, Y 42.092, Z 54.400} C_DIS
   LIN {X -6.695, Y 41.359, Z 54.400} C_DIS
   LIN {X -6.823, Y 40.695, Z 54.400} C_DIS
   LIN {X -6.725, Y 40.156, Z 54.400} C_DIS
   LIN {X -6.567, Y 39.270, Z 54.400} C_DIS
   LIN {X -6.176, Y 38.166, Z 54.400} C_DIS
   LIN {X -6.128, Y 38.030, Z 54.400} C_DIS
   LIN {X -5.636, Y 36.575, Z 54.400} C_DIS
   LIN {X -5.069, Y 34.739, Z 54.400} C_DIS
   LIN {X -4.938, Y 34.309, Z 54.400} C_DIS
   LIN {X -4.772, Y 33.700, Z 54.400} C_DIS
   LIN {X -4.313, Y 32.022, Z 54.400} C_DIS
   LIN {X -4.204, Y 31.571, Z 54.400} C_DIS
   LIN {X -3.996, Y 30.713, Z 54.400} C_DIS
   LIN {X -3.627, Y 29.082, Z 54.400} C_DIS
   LIN {X -2.884, Y 24.933, Z 54.400} C_DIS
   LIN {X -2.805, Y 24.495, Z 54.400} C_DIS
   LIN {X -2.755, Y 24.159, Z 54.400} C_DIS
   LIN {X -2.600, Y 21.478, Z 54.400} C_DIS
   LIN {X -2.200, Y 15.119, Z 54.400} C_DIS
   LIN {X -2.039, Y 12.924, Z 54.400} C_DIS
   LIN {X -2.135, Y 10.889, Z 54.400} C_DIS
   LIN {X -2.577, Y 5.058, Z 54.400} C_DIS
   LIN {X -3.080, Y 1.754, Z 54.400} C_DIS
   LIN {X -3.728, Y -1.666, Z 54.400} C_DIS
   LIN {X -4.414, Y -4.419, Z 54.400} C_DIS
   LIN {X -5.115, Y -7.034, Z 54.400} C_DIS
   LIN {X -5.861, Y -9.297, Z 54.400} C_DIS
   LIN {X -6.363, Y -10.807, Z 54.400} C_DIS
   LIN {X -6.884, Y -12.128, Z 54.400} C_DIS
   LIN {X -7.772, Y -14.405, Z 54.400} C_DIS
   LIN {X -8.342, Y -15.688, Z 54.400} C_DIS
   LIN {X -8.974, Y -17.096, Z 54.400} C_DIS
   LIN {X -9.473, Y -18.918, Z 54.400} C_DIS
   LIN {X -9.805, Y -20.156, Z 54.400} C_DIS
   LIN {X -9.640, Y -21.504, Z 54.400} C_DIS
   LIN {X -9.366, Y -23.840, Z 54.400} C_DIS
   LIN {X -8.356, Y -25.543, Z 54.400} C_DIS
   LIN {X -7.444, Y -27.060, Z 54.400} C_DIS
   LIN {X -5.175, Y -28.811, Z 54.400} C_DIS
   LIN {X 0.502, Y -29.800, Z 54.400} C_DIS
   LIN {X 2.988, Y -28.900, Z 54.400} C_DIS
   LIN {X 3.839, Y -28.572, Z 54.400} C_DIS
   LIN {X 4.854, Y -27.604, Z 54.400} C_DIS
   LIN {X 6.547, Y -26.031, Z 54.400} C_DIS
   LIN {X 7.188, Y -24.536, Z 54.400} C_DIS
   LIN {X 8.034, Y -22.529, Z 54.400} C_DIS
   LIN {X 8.469, Y -20.024, Z 54.400} C_DIS
   LIN {X 8.596, Y -19.314, Z 54.400} C_DIS
   LIN {X 8.682, Y -18.745, Z 54.400} C_DIS
   LIN {X 9.026, Y -16.385, Z 54.400} C_DIS
   LIN {X 9.409, Y -13.089, Z 54.400} C_DIS
   LIN {X 9.462, Y -12.604, Z 54.400} C_DIS
   LIN {X 9.549, Y -11.422, Z 54.400} C_DIS
   LIN {X 9.826, Y -7.829, Z 54.400} C_DIS
   LIN {X 9.901, Y -5.260, Z 54.400} C_DIS
   LIN {X 9.988, Y -1.317, Z 54.400} C_DIS
   LIN {X 9.891, Y 1.677, Z 54.400} C_DIS
   LIN {X 9.845, Y 2.972, Z 54.400} C_DIS
   LIN {X 9.832, Y 3.322, Z 54.400} C_DIS
   LIN {X 9.826, Y 4.259, Z 54.400} C_DIS
   LIN {X 9.558, Y 6.739, Z 54.400} C_DIS
   LIN {X 8.900, Y 13.550, Z 54.400} C_DIS
   LIN {X 7.210, Y 22.416, Z 54.400} C_DIS
   LIN {X 6.627, Y 25.202, Z 54.400} C_DIS
   LIN {X 4.841, Y 31.465, Z 54.400} C_DIS
   LIN {X 4.712, Y 31.861, Z 54.400} C_DIS
   LIN {X 3.802, Y 34.597, Z 54.400} C_DIS
   LIN {X 3.636, Y 35.051, Z 54.400} C_DIS
   LIN {X 2.758, Y 37.463, Z 54.400} C_DIS
   LIN {X 2.335, Y 38.546, Z 54.400} C_DIS
   LIN {X 2.034, Y 39.319, Z 54.400} C_DIS
   LIN {X 1.792, Y 39.912, Z 54.400} C_DIS
   LIN {X 1.409, Y 40.846, Z 54.400} C_DIS
   LIN {X 0.923, Y 41.986, Z 54.400} C_DIS
   LIN {X 0.828, Y 42.212, Z 54.400} C_DIS
   LIN {X 0.726, Y 42.364, Z 54.400} C_DIS
   LIN {X 0.006, Y 43.433, Z 54.400} C_DIS
   LIN {X -1.183, Y 44.207, Z 54.400} C_DIS
   LIN {X -1.453, Y 44.382, Z 54.400}
   LaserEnd_Ext()
   LIN {X 1.541, Y -28.360, Z 54.400}
   LaserStart_Ext()
   LIN {X -1.989, Y -28.360, Z 54.400}
   LaserEnd_Ext()
   LIN {X -5.418, Y -27.360, Z 54.400}
   LaserStart_Ext()
   LIN {X 3.661, Y -27.360, Z 54.400}
   LaserEnd_Ext()
   LIN {X 4.724, Y -26.360, Z 54.400}
   LaserStart_Ext()
   LIN {X 1.402, Y -26.360, Z 54.400}
   LaserEnd_Ext()
   LIN {X -3.226, Y -26.360, Z 54.400}
   LaserStart_Ext()
   LIN {X -6.698, Y -26.360, Z 54.400}
   LaserEnd_Ext()
   LIN {X -7.300, Y -25.360, Z 54.400}
   LaserStart_Ext()
   LIN {X -4.841, Y -25.360, Z 54.400}
   LaserEnd_Ext()
   LIN {X 3.042, Y -25.360, Z 54.400}
   LaserStart_Ext()
   LIN {X 5.747, Y -25.360, Z 54.400}
   LaserEnd_Ext()
   LIN {X 6.175, Y -24.360, Z 54.400}
   LaserStart_Ext()
   LIN {X 3.999, Y -24.360, Z 54.400}
   LaserEnd_Ext()
   LIN {X -5.614, Y -24.360, Z 54.400}
   LaserStart_Ext()
   LIN {X -7.895, Y -24.360, Z 54.400}
   LaserEnd_Ext()
   LIN {X -8.415, Y -23.360, Z 54.400}
   LaserStart_Ext()
   LIN {X -6.299, Y -23.360, Z 54.400}
   LaserEnd_Ext()
   LIN {X 4.445, Y -23.360, Z 54.400}
   LaserStart_Ext()
   LIN {X 6.598, Y -23.360, Z 54.400}
   LaserEnd_Ext()
   LIN {X 7.020, Y -22.360, Z 54.400}
   LaserStart_Ext()
   LIN {X 4.912, Y -22.360, Z 54.400}
   LaserEnd_Ext()
   LIN {X -6.560, Y -22.360, Z 54.400}
   LaserStart_Ext()
   LIN {X -8.533, Y -22.360, Z 54.400}
   LaserEnd_Ext()
   LIN {X -8.650, Y -21.360, Z 54.400}
   LaserStart_Ext()
   LIN {X -6.736, Y -21.360, Z 54.400}
   LaserEnd_Ext()
   LIN {X 5.097, Y -21.360, Z 54.400}
   LaserStart_Ext()
   LIN {X 7.222, Y -21.360, Z 54.400}
   LaserEnd_Ext()
   LIN {X 7.396, Y -20.360, Z 54.400}
   LaserStart_Ext()
   LIN {X 5.038, Y -20.360, Z 54.400}
   LaserEnd_Ext()
   LIN {X -6.748, Y -20.360, Z 54.400}
   LaserStart_Ext()
   LIN {X -8.773, Y -20.360, Z 54.400}
   LaserEnd_Ext()
   LIN {X -8.556, Y -19.360, Z 54.400}
   LaserStart_Ext()
   LIN {X -6.405, Y -19.360, Z 54.400}
   LaserEnd_Ext()
   LIN {X 4.980, Y -19.360, Z 54.400}
   LaserStart_Ext()
   LIN {X 7.572, Y -19.360, Z 54.400}
   LaserEnd_Ext()
   LIN {X 7.728, Y -18.360, Z 54.400}
   LaserStart_Ext()
   LIN {X 4.487, Y -18.360, Z 54.400}
   LaserEnd_Ext()
   LIN {X -6.063, Y -18.360, Z 54.400}
   LaserStart_Ext()
   LIN {X -8.283, Y -18.360, Z 54.400}
   LaserEnd_Ext()
   LIN {X -7.997, Y -17.360, Z 54.400}
   LaserStart_Ext()
   LIN {X -5.656, Y -17.360, Z 54.400}
   LaserEnd_Ext()
   LIN {X 3.885, Y -17.360, Z 54.400}
   LaserStart_Ext()
   LIN {X 7.873, Y -17.360, Z 54.400}
   LaserEnd_Ext()
   LIN {X 8.019, Y -16.360, Z 54.400}
   LaserStart_Ext()
   LIN {X 3.069, Y -16.360, Z 54.400}
   LaserEnd_Ext()
   LIN {X -4.583, Y -16.360, Z 54.400}
   LaserStart_Ext()
   LIN {X -7.547, Y -16.360, Z 54.400}
   LaserEnd_Ext()
   LIN {X -7.102, Y -15.360, Z 54.400}
   LaserStart_Ext()
   LIN {X -2.803, Y -15.360, Z 54.400}
   LaserEnd_Ext()
   LIN {X 1.466, Y -15.360, Z 54.400}
   LaserStart_Ext()
   LIN {X 8.138, Y -15.360, Z 54.400}
   LaserEnd_Ext()
   LIN {X 8.255, Y -14.360, Z 54.400}
   LaserStart_Ext()
   LIN {X -6.682, Y -14.360, Z 54.400}
   LaserEnd_Ext()
   LIN {X -6.291, Y -13.360, Z 54.400}
   LaserStart_Ext()
   LIN {X 8.371, Y -13.360, Z 54.400}
   LaserEnd_Ext()
   LIN {X 8.478, Y -12.360, Z 54.400}
   LaserStart_Ext()
   LIN {X -5.900, Y -12.360, Z 54.400}
   LaserEnd_Ext()
   LIN {X -5.506, Y -11.360, Z 54.400}
   LaserStart_Ext()
   LIN {X 8.551, Y -11.360, Z 54.400}
   LaserEnd_Ext()
   LIN {X 8.628, Y -10.360, Z 54.400}
   LaserStart_Ext()
   LIN {X -5.161, Y -10.360, Z 54.400}
   LaserEnd_Ext()
   LIN {X -4.829, Y -9.360, Z 54.400}
   LaserStart_Ext()
   LIN {X 8.705, Y -9.360, Z 54.400}
   LaserEnd_Ext()
   LIN {X 8.782, Y -8.360, Z 54.400}
   LaserStart_Ext()
   LIN {X -4.499, Y -8.360, Z 54.400}
   LaserEnd_Ext()
   LIN {X -4.169, Y -7.360, Z 54.400}
   LaserStart_Ext()
   LIN {X 8.839, Y -7.360, Z 54.400}
   LaserEnd_Ext()
   LIN {X 8.869, Y -6.360, Z 54.400}
   LaserStart_Ext()
   LIN {X -3.899, Y -6.360, Z 54.400}
   LaserEnd_Ext()
   LIN {X -3.631, Y -5.360, Z 54.400}
   LaserStart_Ext()
   LIN {X 8.898, Y -5.360, Z 54.400}
   LaserEnd_Ext()
   LIN {X 8.921, Y -4.360, Z 54.400}
   LaserStart_Ext()
   LIN {X -3.369, Y -4.360, Z 54.400}
   LaserEnd_Ext()
   LIN {X -3.119, Y -3.360, Z 54.400}
   LaserStart_Ext()
   LIN {X 8.943, Y -3.360, Z 54.400}
   LaserEnd_Ext()
   LIN {X 8.965, Y -2.360, Z 54.400}
   LaserStart_Ext()
   LIN {X -2.870, Y -2.360, Z 54.400}
   LaserEnd_Ext()
   LIN {X -2.652, Y -1.360, Z 54.400}
   LaserStart_Ext()
   LIN {X 8.987, Y -1.360, Z 54.400}
   LaserEnd_Ext()
   LIN {X 8.957, Y -0.360, Z 54.400}
   LaserStart_Ext()
   LIN {X -2.462, Y -0.360, Z 54.400}
   LaserEnd_Ext()
   LIN {X -2.273, Y 0.640, Z 54.400}
   LaserStart_Ext()
   LIN {X 8.924, Y 0.640, Z 54.400}
   LaserEnd_Ext()
   LIN {X 8.892, Y 1.640, Z 54.400}
   LaserStart_Ext()
   LIN {X -2.086, Y 1.640, Z 54.400}
   LaserEnd_Ext()
   LIN {X -1.933, Y 2.640, Z 54.400}
   LaserStart_Ext()
   LIN {X 8.856, Y 2.640, Z 54.400}
   LaserEnd_Ext()
   LIN {X 8.830, Y 3.640, Z 54.400}
   LaserStart_Ext()
   LIN {X -1.781, Y 3.640, Z 54.400}
   LaserEnd_Ext()
   LIN {X -1.629, Y 4.640, Z 54.400}
   LaserStart_Ext()
   LIN {X 8.779, Y 4.640, Z 54.400}
   LaserEnd_Ext()
   LIN {X 8.671, Y 5.640, Z 54.400}
   LaserStart_Ext()
   LIN {X -1.530, Y 5.640, Z 54.400}
   LaserEnd_Ext()
   LIN {X -1.454, Y 6.640, Z 54.400}
   LaserStart_Ext()
   LIN {X 8.563, Y 6.640, Z 54.400}
   LaserEnd_Ext()
   LIN {X 8.466, Y 7.640, Z 54.400}
   LaserStart_Ext()
   LIN {X -1.378, Y 7.640, Z 54.400}
   LaserEnd_Ext()
   LIN {X -1.303, Y 8.640, Z 54.400}
   LaserStart_Ext()
   LIN {X 8.370, Y 8.640, Z 54.400}
   LaserEnd_Ext()
   LIN {X 8.273, Y 9.640, Z 54.400}
   LaserStart_Ext()
   LIN {X -1.227, Y 9.640, Z 54.400}
   LaserEnd_Ext()
   LIN {X -1.151, Y 10.640, Z 54.400}
   LaserStart_Ext()
   LIN {X 8.176, Y 10.640, Z 54.400}
   LaserEnd_Ext()
   LIN {X 8.080, Y 11.640, Z 54.400}
   LaserStart_Ext()
   LIN {X -1.098, Y 11.640, Z 54.400}
   LaserEnd_Ext()
   LIN {X -1.051, Y 12.640, Z 54.400}
   LaserStart_Ext()
   LIN {X 7.983, Y 12.640, Z 54.400}
   LaserEnd_Ext()
   LIN {X 7.865, Y 13.640, Z 54.400}
   LaserStart_Ext()
   LIN {X -1.089, Y 13.640, Z 54.400}
   LaserEnd_Ext()
   LIN {X -1.162, Y 14.640, Z 54.400}
   LaserStart_Ext()
   LIN {X 7.674, Y 14.640, Z 54.400}
   LaserEnd_Ext()
   LIN {X 7.483, Y 15.640, Z 54.400}
   LaserStart_Ext()
   LIN {X -1.231, Y 15.640, Z 54.400}
   LaserEnd_Ext()
   LIN {X -1.294, Y 16.640, Z 54.400}
   LaserStart_Ext()
   LIN {X 7.293, Y 16.640, Z 54.400}
   LaserEnd_Ext()
   LIN {X 7.102, Y 17.640, Z 54.400}
   LaserStart_Ext()
   LIN {X -1.357, Y 17.640, Z 54.400}
   LaserEnd_Ext()
   LIN {X -1.419, Y 18.640, Z 54.400}
   LaserStart_Ext()
   LIN {X 6.912, Y 18.640, Z 54.400}
   LaserEnd_Ext()
   LIN {X 6.721, Y 19.640, Z 54.400}
   LaserStart_Ext()
   LIN {X -1.482, Y 19.640, Z 54.400}
   LaserEnd_Ext()
   LIN {X -1.545, Y 20.640, Z 54.400}
   LaserStart_Ext()
   LIN {X 6.531, Y 20.640, Z 54.400}
   LaserEnd_Ext()
   LIN {X 6.340, Y 21.640, Z 54.400}
   LaserStart_Ext()
   LIN {X -1.607, Y 21.640, Z 54.400}
   LaserEnd_Ext()
   LIN {X -1.665, Y 22.640, Z 54.400}
   LaserStart_Ext()
   LIN {X 6.142, Y 22.640, Z 54.400}
   LaserEnd_Ext()
   LIN {X 5.932, Y 23.640, Z 54.400}
   LaserStart_Ext()
   LIN {X -1.723, Y 23.640, Z 54.400}
   LaserEnd_Ext()
   LIN {X -1.816, Y 24.640, Z 54.400}
   LaserStart_Ext()
   LIN {X 5.723, Y 24.640, Z 54.400}
   LaserEnd_Ext()
   LIN {X 5.462, Y 25.640, Z 54.400}
   LaserStart_Ext()
   LIN {X -1.995, Y 25.640, Z 54.400}
   LaserEnd_Ext()
   LIN {X -2.174, Y 26.640, Z 54.400}
   LaserStart_Ext()
   LIN {X 5.177, Y 26.640, Z 54.400}
   LaserEnd_Ext()
   LIN {X 4.892, Y 27.640, Z 54.400}
   LaserStart_Ext()
   LIN {X -2.353, Y 27.640, Z 54.400}
   LaserEnd_Ext()
   LIN {X -2.532, Y 28.640, Z 54.400}
   LaserStart_Ext()
   LIN {X 4.607, Y 28.640, Z 54.400}
   LaserEnd_Ext()
   LIN {X 4.322, Y 29.640, Z 54.400}
   LaserStart_Ext()
   LIN {X -2.728, Y 29.640, Z 54.400}
   LaserEnd_Ext()
   LIN {X -2.954, Y 30.640, Z 54.400}
   LaserStart_Ext()
   LIN {X 4.037, Y 30.640, Z 54.400}
   LaserEnd_Ext()
   LIN {X 3.731, Y 31.640, Z 54.400}
   LaserStart_Ext()
   LIN {X -3.192, Y 31.640, Z 54.400}
   LaserEnd_Ext()
   LIN {X -3.446, Y 32.640, Z 54.400}
   LaserStart_Ext()
   LIN {X 3.399, Y 32.640, Z 54.400}
   LaserEnd_Ext()
   LIN {X 3.066, Y 33.640, Z 54.400}
   LaserStart_Ext()
   LIN {X -3.719, Y 33.640, Z 54.400}
   LaserEnd_Ext()
   LIN {X -3.993, Y 34.640, Z 54.400}
   LaserStart_Ext()
   LIN {X 2.722, Y 34.640, Z 54.400}
   LaserEnd_Ext()
   LIN {X 2.358, Y 35.640, Z 54.400}
   LaserStart_Ext()
   LIN {X -4.301, Y 35.640, Z 54.400}
   LaserEnd_Ext()
   LIN {X -4.610, Y 36.640, Z 54.400}
   LaserStart_Ext()
   LIN {X 1.994, Y 36.640, Z 54.400}
   LaserEnd_Ext()
   LIN {X 1.615, Y 37.640, Z 54.400}
   LaserStart_Ext()
   LIN {X -4.941, Y 37.640, Z 54.400}
   LaserEnd_Ext()
   LIN {X -5.283, Y 38.640, Z 54.400}
   LaserStart_Ext()
   LIN {X 1.225, Y 38.640, Z 54.400}
   LaserEnd_Ext()
   LIN {X 0.823, Y 39.640, Z 54.400}
   LaserStart_Ext()
   LIN {X -5.617, Y 39.640, Z 54.400}
   LaserEnd_Ext()
   LIN {X -5.796, Y 40.640, Z 54.400}
   LaserStart_Ext()
   LIN {X 0.410, Y 40.640, Z 54.400}
   LaserEnd_Ext()
   LIN {X -0.016, Y 41.640, Z 54.400}
   LaserStart_Ext()
   LIN {X -5.626, Y 41.640, Z 54.400}
   LaserEnd_Ext()
   LIN {X -5.039, Y 42.640, Z 54.400}
   LaserStart_Ext()
   LIN {X -0.666, Y 42.640, Z 54.400}
   LaserEnd_Ext()
   LIN {X 0.941, Y -16.115, Z 55.250}
   LaserStart_Ext()
   LIN {X 1.476, Y -16.445, Z 55.250} C_DIS
   LIN {X 2.747, Y -17.235, Z 55.250} C_DIS
   LIN {X 3.667, Y -18.761, Z 55.250} C_DIS
   LIN {X 4.062, Y -19.411, Z 55.250} C_DIS
   LIN {X 4.101, Y -20.032, Z 55.250} C_DIS
   LIN {X 4.194, Y -21.618, Z 55.250} C_DIS
   LIN {X 3.609, Y -22.993, Z 55.250} C_DIS
   LIN {X 3.127, Y -23.981, Z 55.250} C_DIS
   LIN {X 1.829, Y -25.084, Z 55.250} C_DIS
   LIN {X 1.686, Y -25.203, Z 55.250} C_DIS
   LIN {X 1.588, Y -25.232, Z 55.250} C_DIS
   LIN {X -0.415, Y -25.832, Z 55.250} C_DIS
   LIN {X -1.748, Y -25.659, Z 55.250} C_DIS
   LIN {X -2.443, Y -25.566, Z 55.250} C_DIS
   LIN {X -3.238, Y -25.076, Z 55.250} C_DIS
   LIN {X -4.203, Y -24.484, Z 55.250} C_DIS
   LIN {X -4.706, Y -23.756, Z 55.250} C_DIS
   LIN {X -5.383, Y -22.768, Z 55.250} C_DIS
   LIN {X -5.604, Y -21.516, Z 55.250} C_DIS
   LIN {X -5.748, Y -20.714, Z 55.250} C_DIS
   LIN {X -5.516, Y -20.021, Z 55.250} C_DIS
   LIN {X -4.808, Y -17.946, Z 55.250} C_DIS
   LIN {X -3.307, Y -16.565, Z 55.250} C_DIS
   LIN {X -1.191, Y -15.861, Z 55.250} C_DIS
   LIN {X 0.412, Y -16.053, Z 55.250} C_DIS
   LIN {X 0.941, Y -16.115, Z 55.250}
   LaserEnd_Ext()
   LIN {X -5.644, Y 43.549, Z 55.250}
   LaserStart_Ext()
   LIN {X -5.877, Y 43.356, Z 55.250} C_DIS
   LIN {X -6.205, Y 42.822, Z 55.250} C_DIS
   LIN {X -6.617, Y 42.158, Z 55.250} C_DIS
   LIN {X -6.752, Y 41.449, Z 55.250} C_DIS
   LIN {X -6.889, Y 40.732, Z 55.250} C_DIS
   LIN {X -6.727, Y 39.840, Z 55.250} C_DIS
   LIN {X -6.630, Y 39.307, Z 55.250} C_DIS
   LIN {X -6.520, Y 39.001, Z 55.250} C_DIS
   LIN {X -6.210, Y 38.129, Z 55.250} C_DIS
   LIN {X -5.746, Y 36.770, Z 55.250} C_DIS
   LIN {X -5.693, Y 36.614, Z 55.250} C_DIS
   LIN {X -5.603, Y 36.322, Z 55.250} C_DIS
   LIN {X -4.989, Y 34.350, Z 55.250} C_DIS
   LIN {X -4.570, Y 32.835, Z 55.250} C_DIS
   LIN {X -4.359, Y 32.064, Z 55.250} C_DIS
   LIN {X -4.045, Y 30.766, Z 55.250} C_DIS
   LIN {X -3.914, Y 30.226, Z 55.250} C_DIS
   LIN {X -3.683, Y 29.201, Z 55.250} C_DIS
   LIN {X -2.956, Y 25.144, Z 55.250} C_DIS
   LIN {X -2.772, Y 24.130, Z 55.250} C_DIS
   LIN {X -2.282, Y 16.333, Z 55.250} C_DIS
   LIN {X -2.040, Y 13.054, Z 55.250} C_DIS
   LIN {X -2.185, Y 10.012, Z 55.250} C_DIS
   LIN {X -2.550, Y 5.186, Z 55.250} C_DIS
   LIN {X -3.161, Y 1.176, Z 55.250} C_DIS
   LIN {X -3.655, Y -1.434, Z 55.250} C_DIS
   LIN {X -4.641, Y -5.387, Z 55.250} C_DIS
   LIN {X -5.086, Y -7.048, Z 55.250} C_DIS
   LIN {X -6.101, Y -10.126, Z 55.250} C_DIS
   LIN {X -6.321, Y -10.802, Z 55.250} C_DIS
   LIN {X -6.552, Y -11.405, Z 55.250} C_DIS
   LIN {X -7.711, Y -14.372, Z 55.250} C_DIS
   LIN {X -8.812, Y -16.856, Z 55.250} C_DIS
   LIN {X -8.906, Y -17.064, Z 55.250} C_DIS
   LIN {X -8.980, Y -17.334, Z 55.250} C_DIS
   LIN {X -9.729, Y -20.126, Z 55.250} C_DIS
   LIN {X -9.356, Y -23.167, Z 55.250} C_DIS
   LIN {X -9.281, Y -23.809, Z 55.250} C_DIS
   LIN {X -9.004, Y -24.277, Z 55.250} C_DIS
   LIN {X -7.352, Y -27.024, Z 55.250} C_DIS
   LIN {X -5.871, Y -28.167, Z 55.250} C_DIS
   LIN {X -5.046, Y -28.795, Z 55.250} C_DIS
   LIN {X -4.642, Y -28.976, Z 55.250} C_DIS
   LIN {X -2.860, Y -29.165, Z 55.250} C_DIS
   LIN {X 0.570, Y -29.751, Z 55.250} C_DIS
   LIN {X 2.070, Y -29.207, Z 55.250} C_DIS
   LIN {X 4.014, Y -28.459, Z 55.250} C_DIS
   LIN {X 6.332, Y -26.248, Z 55.250} C_DIS
   LIN {X 6.634, Y -25.967, Z 55.250} C_DIS
   LIN {X 6.748, Y -25.700, Z 55.250} C_DIS
   LIN {X 8.116, Y -22.457, Z 55.250} C_DIS
   LIN {X 8.562, Y -19.886, Z 55.250} C_DIS
   LIN {X 8.670, Y -19.241, Z 55.250} C_DIS
   LIN {X 8.775, Y -18.495, Z 55.250} C_DIS
   LIN {X 9.093, Y -16.310, Z 55.250} C_DIS
   LIN {X 9.328, Y -14.290, Z 55.250} C_DIS
   LIN {X 9.521, Y -12.528, Z 55.250} C_DIS
   LIN {X 9.836, Y -8.235, Z 55.250} C_DIS
   LIN {X 9.873, Y -7.752, Z 55.250} C_DIS
   LIN {X 9.883, Y -7.408, Z 55.250} C_DIS
   LIN {X 10.020, Y -1.240, Z 55.250} C_DIS
   LIN {X 9.868, Y 3.443, Z 55.250} C_DIS
   LIN {X 9.854, Y 3.829, Z 55.250} C_DIS
   LIN {X 9.850, Y 3.933, Z 55.250} C_DIS
   LIN {X 9.849, Y 4.213, Z 55.250} C_DIS
   LIN {X 9.769, Y 4.952, Z 55.250} C_DIS
   LIN {X 9.000, Y 12.909, Z 55.250} C_DIS
   LIN {X 7.026, Y 23.267, Z 55.250} C_DIS
   LIN {X 6.659, Y 25.020, Z 55.250} C_DIS
   LIN {X 5.514, Y 29.036, Z 55.250} C_DIS
   LIN {X 4.886, Y 31.251, Z 55.250} C_DIS
   LIN {X 4.282, Y 33.071, Z 55.250} C_DIS
   LIN {X 3.829, Y 34.432, Z 55.250} C_DIS
   LIN {X 3.039, Y 36.598, Z 55.250} C_DIS
   LIN {X 2.784, Y 37.298, Z 55.250} C_DIS
   LIN {X 2.458, Y 38.133, Z 55.250} C_DIS
   LIN {X 2.010, Y 39.277, Z 55.250} C_DIS
   LIN {X 1.560, Y 40.371, Z 55.250} C_DIS
   LIN {X 1.342, Y 40.902, Z 55.250} C_DIS
   LIN {X 1.204, Y 41.227, Z 55.250} C_DIS
   LIN {X 0.757, Y 42.267, Z 55.250} C_DIS
   LIN {X -0.053, Y 43.465, Z 55.250} C_DIS
   LIN {X -1.528, Y 44.431, Z 55.250} C_DIS
   LIN {X -2.747, Y 44.598, Z 55.250} C_DIS
   LIN {X -3.258, Y 44.667, Z 55.250} C_DIS
   LIN {X -4.464, Y 44.068, Z 55.250} C_DIS
   LIN {X -5.644, Y 43.549, Z 55.250}
   LaserEnd_Ext()
   LIN {X 8.602, Y 6.631, Z 55.250}
   LaserStart_Ext()
   LIN {X 8.602, Y -11.389, Z 55.250}
   LaserEnd_Ext()
   LIN {X 7.602, Y -19.566, Z 55.250}
   LaserStart_Ext()
   LIN {X 7.602, Y 14.901, Z 55.250}
   LaserEnd_Ext()
   LIN {X 6.602, Y 20.149, Z 55.250}
   LaserStart_Ext()
   LIN {X 6.602, Y -23.473, Z 55.250}
   LaserEnd_Ext()
   LIN {X 5.602, Y -25.562, Z 55.250}
   LaserStart_Ext()
   LIN {X 5.602, Y 25.079, Z 55.250}
   LaserEnd_Ext()
   LIN {X 4.602, Y 28.587, Z 55.250}
   LaserStart_Ext()
   LIN {X 4.602, Y -18.374, Z 55.250}
   LaserEnd_Ext()
   LIN {X 4.602, Y -23.213, Z 55.250}
   LaserStart_Ext()
   LIN {X 4.602, Y -26.516, Z 55.250}
   LaserEnd_Ext()
   LIN {X 3.602, Y -27.470, Z 55.250}
   LaserStart_Ext()
   LIN {X 3.602, Y -24.890, Z 55.250}
   LaserEnd_Ext()
   LIN {X 3.602, Y -16.717, Z 55.250}
   LaserStart_Ext()
   LIN {X 3.602, Y 31.944, Z 55.250}
   LaserEnd_Ext()
   LIN {X 2.602, Y 34.878, Z 55.250}
   LaserStart_Ext()
   LIN {X 2.602, Y -15.967, Z 55.250}
   LaserEnd_Ext()
   LIN {X 2.602, Y -25.739, Z 55.250}
   LaserStart_Ext()
   LIN {X 2.602, Y -27.931, Z 55.250}
   LaserEnd_Ext()
   LIN {X 1.602, Y -28.313, Z 55.250}
   LaserStart_Ext()
   LIN {X 1.602, Y -26.272, Z 55.250}
   LaserEnd_Ext()
   LIN {X 1.602, Y -15.347, Z 55.250}
   LaserStart_Ext()
   LIN {X 1.602, Y 37.576, Z 55.250}
   LaserEnd_Ext()
   LIN {X 0.602, Y 40.071, Z 55.250}
   LaserStart_Ext()
   LIN {X 0.602, Y -15.068, Z 55.250}
   LaserEnd_Ext()
   LIN {X 0.602, Y -26.571, Z 55.250}
   LaserStart_Ext()
   LIN {X 0.602, Y -28.675, Z 55.250}
   LaserEnd_Ext()
   LIN {X -0.398, Y -28.571, Z 55.250}
   LaserStart_Ext()
   LIN {X -0.398, Y -26.831, Z 55.250}
   LaserEnd_Ext()
   LIN {X -0.398, Y -14.949, Z 55.250}
   LaserStart_Ext()
   LIN {X -0.398, Y 42.190, Z 55.250}
   LaserEnd_Ext()
   LIN {X -1.398, Y 43.156, Z 55.250}
   LaserStart_Ext()
   LIN {X -1.398, Y 18.217, Z 55.250}
   LaserEnd_Ext()
   LIN {X -1.398, Y 7.156, Z 55.250}
   LaserStart_Ext()
   LIN {X -1.398, Y -14.883, Z 55.250}
   LaserEnd_Ext()
   LIN {X -1.398, Y -26.713, Z 55.250}
   LaserStart_Ext()
   LIN {X -1.398, Y -28.400, Z 55.250}
   LaserEnd_Ext()
   LIN {X -2.398, Y -28.229, Z 55.250}
   LaserStart_Ext()
   LIN {X -2.398, Y -26.581, Z 55.250}
   LaserEnd_Ext()
   LIN {X -2.398, Y -15.202, Z 55.250}
   LaserStart_Ext()
   LIN {X -2.398, Y -0.171, Z 55.250}
   LaserEnd_Ext()
   LIN {X -2.398, Y 27.701, Z 55.250}
   LaserStart_Ext()
   LIN {X -2.398, Y 43.541, Z 55.250}
   LaserEnd_Ext()
   LIN {X -3.398, Y 43.481, Z 55.250}
   LaserStart_Ext()
   LIN {X -3.398, Y 32.340, Z 55.250}
   LaserEnd_Ext()
   LIN {X -3.398, Y -4.536, Z 55.250}
   LaserStart_Ext()
   LIN {X -3.398, Y -15.527, Z 55.250}
   LaserEnd_Ext()
   LIN {X -3.398, Y -26.152, Z 55.250}
   LaserStart_Ext()
   LIN {X -3.398, Y -28.102, Z 55.250}
   LaserEnd_Ext()
   LIN {X -4.398, Y -27.990, Z 55.250}
   LaserStart_Ext()
   LIN {X -4.398, Y -25.538, Z 55.250}
   LaserEnd_Ext()
   LIN {X -4.398, Y -16.210, Z 55.250}
   LaserStart_Ext()
   LIN {X -4.398, Y -8.155, Z 55.250}
   LaserEnd_Ext()
   LIN {X -4.398, Y 35.816, Z 55.250}
   LaserStart_Ext()
   LIN {X -4.398, Y 43.004, Z 55.250}
   LaserEnd_Ext()
   LIN {X -5.398, Y 42.226, Z 55.250}
   LaserStart_Ext()
   LIN {X -5.398, Y 38.831, Z 55.250}
   LaserEnd_Ext()
   LIN {X -5.398, Y -11.189, Z 55.250}
   LaserStart_Ext()
   LIN {X -5.398, Y -17.130, Z 55.250}
   LaserEnd_Ext()
   LIN {X -5.398, Y -24.514, Z 55.250}
   LaserStart_Ext()
   LIN {X -5.398, Y -27.269, Z 55.250}
   LaserEnd_Ext()
   LIN {X -6.398, Y -26.497, Z 55.250}
   LaserStart_Ext()
   LIN {X -6.398, Y -22.773, Z 55.250}
   LaserEnd_Ext()
   LIN {X -6.398, Y -19.510, Z 55.250}
   LaserStart_Ext()
   LIN {X -6.398, Y -13.759, Z 55.250}
   LaserEnd_Ext()
   LIN {X -7.398, Y -16.134, Z 55.250}
   LaserStart_Ext()
   LIN {X -7.398, Y -25.007, Z 55.250}
   LaserEnd_Ext()
   LIN {X -8.398, Y -22.767, Z 55.250}
   LaserStart_Ext()
   LIN {X -8.398, Y -19.025, Z 55.250}
   LaserEnd_Ext()
   LIN {X 3.200, Y -23.888, Z 56.100}
   LaserStart_Ext()
   LIN {X 1.769, Y -25.149, Z 56.100} C_DIS
   LIN {X 0.590, Y -25.506, Z 56.100} C_DIS
   LIN {X -0.325, Y -25.780, Z 56.100} C_DIS
   LIN {X -1.574, Y -25.618, Z 56.100} C_DIS
   LIN {X -2.354, Y -25.519, Z 56.100} C_DIS
   LIN {X -2.848, Y -25.219, Z 56.100} C_DIS
   LIN {X -4.117, Y -24.441, Z 56.100} C_DIS
   LIN {X -5.199, Y -22.875, Z 56.100} C_DIS
   LIN {X -5.301, Y -22.728, Z 56.100} C_DIS
   LIN {X -5.334, Y -22.546, Z 56.100} C_DIS
   LIN {X -5.671, Y -20.674, Z 56.100} C_DIS
   LIN {X -5.030, Y -18.766, Z 56.100} C_DIS
   LIN {X -4.736, Y -17.902, Z 56.100} C_DIS
   LIN {X -4.091, Y -17.309, Z 56.100} C_DIS
   LIN {X -3.211, Y -16.494, Z 56.100} C_DIS
   LIN {X -1.534, Y -15.945, Z 56.100} C_DIS
   LIN {X -1.119, Y -15.811, Z 56.100} C_DIS
   LIN {X -0.807, Y -15.848, Z 56.100} C_DIS
   LIN {X 1.008, Y -16.059, Z 56.100} C_DIS
   LIN {X 2.794, Y -17.162, Z 56.100} C_DIS
   LIN {X 4.137, Y -19.349, Z 56.100} C_DIS
   LIN {X 4.268, Y -21.449, Z 56.100} C_DIS
   LIN {X 4.274, Y -21.555, Z 56.100} C_DIS
   LIN {X 3.356, Y -23.710, Z 56.100} C_DIS
   LIN {X 3.200, Y -23.888, Z 56.100}
   LaserEnd_Ext()
   LIN {X -3.241, Y 0.599, Z 56.100}
   LaserStart_Ext()
   LIN {X -2.524, Y 5.314, Z 56.100} C_DIS
   LIN {X -2.234, Y 9.136, Z 56.100} C_DIS
   LIN {X -2.042, Y 13.183, Z 56.100} C_DIS
   LIN {X -2.363, Y 17.547, Z 56.100} C_DIS
   LIN {X -2.765, Y 23.947, Z 56.100} C_DIS
   LIN {X -3.441, Y 27.661, Z 56.100} C_DIS
   LIN {X -3.738, Y 29.320, Z 56.100} C_DIS
   LIN {X -3.833, Y 29.739, Z 56.100} C_DIS
   LIN {X -3.886, Y 29.960, Z 56.100} C_DIS
   LIN {X -4.406, Y 32.107, Z 56.100} C_DIS
   LIN {X -4.924, Y 33.966, Z 56.100} C_DIS
   LIN {X -5.041, Y 34.391, Z 56.100} C_DIS
   LIN {X -5.134, Y 34.692, Z 56.100} C_DIS
   LIN {X -5.750, Y 36.654, Z 56.100} C_DIS
   LIN {X -6.223, Y 38.032, Z 56.100} C_DIS
   LIN {X -6.270, Y 38.167, Z 56.100} C_DIS
   LIN {X -6.330, Y 38.334, Z 56.100} C_DIS
   LIN {X -6.693, Y 39.344, Z 56.100} C_DIS
   LIN {X -6.842, Y 40.157, Z 56.100} C_DIS
   LIN {X -6.956, Y 40.768, Z 56.100} C_DIS
   LIN {X -6.815, Y 41.522, Z 56.100} C_DIS
   LIN {X -6.687, Y 42.196, Z 56.100} C_DIS
   LIN {X -6.362, Y 42.718, Z 56.100} C_DIS
   LIN {X -5.898, Y 43.452, Z 56.100} C_DIS
   LIN {X -4.973, Y 43.897, Z 56.100} C_DIS
   LIN {X -3.334, Y 44.712, Z 56.100} C_DIS
   LIN {X -1.766, Y 44.501, Z 56.100} C_DIS
   LIN {X -1.604, Y 44.480, Z 56.100} C_DIS
   LIN {X -1.483, Y 44.403, Z 56.100} C_DIS
   LIN {X -0.140, Y 43.538, Z 56.100} C_DIS
   LIN {X 0.625, Y 42.413, Z 56.100} C_DIS
   LIN {X 0.687, Y 42.321, Z 56.100} C_DIS
   LIN {X 0.746, Y 42.183, Z 56.100} C_DIS
   LIN {X 1.275, Y 40.958, Z 56.100} C_DIS
   LIN {X 1.714, Y 39.898, Z 56.100} C_DIS
   LIN {X 1.987, Y 39.235, Z 56.100} C_DIS
   LIN {X 2.347, Y 38.315, Z 56.100} C_DIS
   LIN {X 2.811, Y 37.133, Z 56.100} C_DIS
   LIN {X 3.705, Y 34.681, Z 56.100} C_DIS
   LIN {X 3.864, Y 34.246, Z 56.100} C_DIS
   LIN {X 4.307, Y 32.910, Z 56.100} C_DIS
   LIN {X 4.942, Y 30.997, Z 56.100} C_DIS
   LIN {X 6.220, Y 26.488, Z 56.100} C_DIS
   LIN {X 6.691, Y 24.838, Z 56.100} C_DIS
   LIN {X 6.841, Y 24.117, Z 56.100} C_DIS
   LIN {X 9.099, Y 12.268, Z 56.100} C_DIS
   LIN {X 9.584, Y 7.257, Z 56.100} C_DIS
   LIN {X 9.864, Y 4.300, Z 56.100} C_DIS
   LIN {X 9.888, Y 3.885, Z 56.100} C_DIS
   LIN {X 9.898, Y 3.599, Z 56.100} C_DIS
   LIN {X 10.009, Y 0.170, Z 56.100} C_DIS
   LIN {X 10.052, Y -1.163, Z 56.100} C_DIS
   LIN {X 10.026, Y -2.351, Z 56.100} C_DIS
   LIN {X 9.921, Y -7.676, Z 56.100} C_DIS
   LIN {X 9.829, Y -9.060, Z 56.100} C_DIS
   LIN {X 9.579, Y -12.452, Z 56.100} C_DIS
   LIN {X 9.247, Y -15.492, Z 56.100} C_DIS
   LIN {X 9.161, Y -16.235, Z 56.100} C_DIS
   LIN {X 9.043, Y -17.040, Z 56.100} C_DIS
   LIN {X 8.744, Y -19.167, Z 56.100} C_DIS
   LIN {X 8.437, Y -21.006, Z 56.100} C_DIS
   LIN {X 8.198, Y -22.384, Z 56.100} C_DIS
   LIN {X 7.315, Y -24.478, Z 56.100} C_DIS
   LIN {X 6.803, Y -25.770, Z 56.100} C_DIS
   LIN {X 5.997, Y -26.621, Z 56.100} C_DIS
   LIN {X 4.188, Y -28.346, Z 56.100} C_DIS
   LIN {X 1.152, Y -29.515, Z 56.100} C_DIS
   LIN {X 0.637, Y -29.701, Z 56.100} C_DIS
   LIN {X -0.539, Y -29.500, Z 56.100} C_DIS
   LIN {X -4.133, Y -29.120, Z 56.100} C_DIS
   LIN {X -4.950, Y -28.753, Z 56.100} C_DIS
   LIN {X -6.613, Y -27.487, Z 56.100} C_DIS
   LIN {X -7.260, Y -26.989, Z 56.100} C_DIS
   LIN {X -8.332, Y -25.205, Z 56.100} C_DIS
   LIN {X -9.196, Y -23.778, Z 56.100} C_DIS
   LIN {X -9.354, Y -22.533, Z 56.100} C_DIS
   LIN {X -9.653, Y -20.096, Z 56.100} C_DIS
   LIN {X -9.164, Y -18.274, Z 56.100} C_DIS
   LIN {X -8.837, Y -17.032, Z 56.100} C_DIS
   LIN {X -8.285, Y -15.774, Z 56.100} C_DIS
   LIN {X -7.649, Y -14.339, Z 56.100} C_DIS
   LIN {X -7.087, Y -12.899, Z 56.100} C_DIS
   LIN {X -6.267, Y -10.766, Z 56.100} C_DIS
   LIN {X -5.489, Y -8.371, Z 56.100} C_DIS
   LIN {X -5.057, Y -7.061, Z 56.100} C_DIS
   LIN {X -4.867, Y -6.355, Z 56.100} C_DIS
   LIN {X -3.583, Y -1.202, Z 56.100} C_DIS
   LIN {X -3.241, Y 0.599, Z 56.100}
   LaserEnd_Ext()
   LIN {X -3.482, Y 43.522, Z 56.100}
   LaserStart_Ext()
   LIN {X -1.983, Y 43.522, Z 56.100}
   LaserEnd_Ext()
   LIN {X -0.658, Y 42.522, Z 56.100}
   LaserStart_Ext()
   LIN {X -5.303, Y 42.522, Z 56.100}
   LaserEnd_Ext()
   LIN {X -5.797, Y 41.522, Z 56.100}
   LaserStart_Ext()
   LIN {X -0.057, Y 41.522, Z 56.100}
   LaserEnd_Ext()
   LIN {X 0.373, Y 40.522, Z 56.100}
   LaserStart_Ext()
   LIN {X -5.892, Y 40.522, Z 56.100}
   LaserEnd_Ext()
   LIN {X -5.694, Y 39.522, Z 56.100}
   LaserStart_Ext()
   LIN {X 0.788, Y 39.522, Z 56.100}
   LaserEnd_Ext()
   LIN {X 1.193, Y 38.522, Z 56.100}
   LaserStart_Ext()
   LIN {X -5.335, Y 38.522, Z 56.100}
   LaserEnd_Ext()
   LIN {X -4.991, Y 37.522, Z 56.100}
   LaserStart_Ext()
   LIN {X 1.585, Y 37.522, Z 56.100}
   LaserEnd_Ext()
   LIN {X 1.970, Y 36.522, Z 56.100}
   LaserStart_Ext()
   LIN {X -4.661, Y 36.522, Z 56.100}
   LaserEnd_Ext()
   LIN {X -4.347, Y 35.522, Z 56.100}
   LaserStart_Ext()
   LIN {X 2.334, Y 35.522, Z 56.100}
   LaserEnd_Ext()
   LIN {X 2.699, Y 34.522, Z 56.100}
   LaserStart_Ext()
   LIN {X -4.040, Y 34.522, Z 56.100}
   LaserEnd_Ext()
   LIN {X -3.762, Y 33.522, Z 56.100}
   LaserStart_Ext()
   LIN {X 3.050, Y 33.522, Z 56.100}
   LaserEnd_Ext()
   LIN {X 3.382, Y 32.522, Z 56.100}
   LaserStart_Ext()
   LIN {X -3.483, Y 32.522, Z 56.100}
   LaserEnd_Ext()
   LIN {X -3.235, Y 31.522, Z 56.100}
   LaserStart_Ext()
   LIN {X 3.714, Y 31.522, Z 56.100}
   LaserEnd_Ext()
   LIN {X 4.037, Y 30.522, Z 56.100}
   LaserStart_Ext()
   LIN {X -2.993, Y 30.522, Z 56.100}
   LaserEnd_Ext()
   LIN {X -2.759, Y 29.522, Z 56.100}
   LaserStart_Ext()
   LIN {X 4.321, Y 29.522, Z 56.100}
   LaserEnd_Ext()
   LIN {X 4.604, Y 28.522, Z 56.100}
   LaserStart_Ext()
   LIN {X -2.579, Y 28.522, Z 56.100}
   LaserEnd_Ext()
   LIN {X -2.399, Y 27.522, Z 56.100}
   LaserStart_Ext()
   LIN {X 4.888, Y 27.522, Z 56.100}
   LaserEnd_Ext()
   LIN {X 5.171, Y 26.522, Z 56.100}
   LaserStart_Ext()
   LIN {X -2.217, Y 26.522, Z 56.100}
   LaserEnd_Ext()
   LIN {X -2.035, Y 25.522, Z 56.100}
   LaserStart_Ext()
   LIN {X 5.456, Y 25.522, Z 56.100}
   LaserEnd_Ext()
   LIN {X 5.735, Y 24.522, Z 56.100}
   LaserStart_Ext()
   LIN {X -1.853, Y 24.522, Z 56.100}
   LaserEnd_Ext()
   LIN {X -1.737, Y 23.522, Z 56.100}
   LaserStart_Ext()
   LIN {X 5.937, Y 23.522, Z 56.100}
   LaserEnd_Ext()
   LIN {X 6.127, Y 22.522, Z 56.100}
   LaserStart_Ext()
   LIN {X -1.674, Y 22.522, Z 56.100}
   LaserEnd_Ext()
   LIN {X -1.611, Y 21.522, Z 56.100}
   LaserStart_Ext()
   LIN {X 6.318, Y 21.522, Z 56.100}
   LaserEnd_Ext()
   LIN {X 6.509, Y 20.522, Z 56.100}
   LaserStart_Ext()
   LIN {X -1.548, Y 20.522, Z 56.100}
   LaserEnd_Ext()
   LIN {X -1.485, Y 19.522, Z 56.100}
   LaserStart_Ext()
   LIN {X 6.699, Y 19.522, Z 56.100}
   LaserEnd_Ext()
   LIN {X 6.890, Y 18.522, Z 56.100}
   LaserStart_Ext()
   LIN {X -1.423, Y 18.522, Z 56.100}
   LaserEnd_Ext()
   LIN {X -1.359, Y 17.522, Z 56.100}
   LaserStart_Ext()
   LIN {X 7.080, Y 17.522, Z 56.100}
   LaserEnd_Ext()
   LIN {X 7.271, Y 16.522, Z 56.100}
   LaserStart_Ext()
   LIN {X -1.285, Y 16.522, Z 56.100}
   LaserEnd_Ext()
   LIN {X -1.212, Y 15.522, Z 56.100}
   LaserStart_Ext()
   LIN {X 7.461, Y 15.522, Z 56.100}
   LaserEnd_Ext()
   LIN {X 7.652, Y 14.522, Z 56.100}
   LaserStart_Ext()
   LIN {X -1.138, Y 14.522, Z 56.100}
   LaserEnd_Ext()
   LIN {X -1.065, Y 13.522, Z 56.100}
   LaserStart_Ext()
   LIN {X 7.843, Y 13.522, Z 56.100}
   LaserEnd_Ext()
   LIN {X 8.033, Y 12.522, Z 56.100}
   LaserStart_Ext()
   LIN {X -1.073, Y 12.522, Z 56.100}
   LaserEnd_Ext()
   LIN {X -1.120, Y 11.522, Z 56.100}
   LaserStart_Ext()
   LIN {X 8.167, Y 11.522, Z 56.100}
   LaserEnd_Ext()
   LIN {X 8.264, Y 10.522, Z 56.100}
   LaserStart_Ext()
   LIN {X -1.167, Y 10.522, Z 56.100}
   LaserEnd_Ext()
   LIN {X -1.215, Y 9.522, Z 56.100}
   LaserStart_Ext()
   LIN {X 8.360, Y 9.522, Z 56.100}
   LaserEnd_Ext()
   LIN {X 8.457, Y 8.522, Z 56.100}
   LaserStart_Ext()
   LIN {X -1.278, Y 8.522, Z 56.100}
   LaserEnd_Ext()
   LIN {X -1.354, Y 7.522, Z 56.100}
   LaserStart_Ext()
   LIN {X 8.554, Y 7.522, Z 56.100}
   LaserEnd_Ext()
   LIN {X 8.649, Y 6.522, Z 56.100}
   LaserStart_Ext()
   LIN {X -1.429, Y 6.522, Z 56.100}
   LaserEnd_Ext()
   LIN {X -1.505, Y 5.522, Z 56.100}
   LaserStart_Ext()
   LIN {X 8.744, Y 5.522, Z 56.100}
   LaserEnd_Ext()
   LIN {X 8.839, Y 4.522, Z 56.100}
   LaserStart_Ext()
   LIN {X -1.633, Y 4.522, Z 56.100}
   LaserEnd_Ext()
   LIN {X -1.785, Y 3.522, Z 56.100}
   LaserStart_Ext()
   LIN {X 8.899, Y 3.522, Z 56.100}
   LaserEnd_Ext()
   LIN {X 8.932, Y 2.522, Z 56.100}
   LaserStart_Ext()
   LIN {X -1.937, Y 2.522, Z 56.100}
   LaserEnd_Ext()
   LIN {X -2.089, Y 1.522, Z 56.100}
   LaserStart_Ext()
   LIN {X 8.964, Y 1.522, Z 56.100}
   LaserEnd_Ext()
   LIN {X 8.997, Y 0.522, Z 56.100}
   LaserStart_Ext()
   LIN {X -2.242, Y 0.522, Z 56.100}
   LaserEnd_Ext()
   LIN {X -2.428, Y -0.478, Z 56.100}
   LaserStart_Ext()
   LIN {X 9.029, Y -0.478, Z 56.100}
   LaserEnd_Ext()
   LIN {X 9.045, Y -1.478, Z 56.100}
   LaserStart_Ext()
   LIN {X -2.621, Y -1.478, Z 56.100}
   LaserEnd_Ext()
   LIN {X -2.870, Y -2.478, Z 56.100}
   LaserStart_Ext()
   LIN {X 9.023, Y -2.478, Z 56.100}
   LaserEnd_Ext()
   LIN {X 9.003, Y -3.478, Z 56.100}
   LaserStart_Ext()
   LIN {X -3.120, Y -3.478, Z 56.100}
   LaserEnd_Ext()
   LIN {X -3.369, Y -4.478, Z 56.100}
   LaserStart_Ext()
   LIN {X 8.984, Y -4.478, Z 56.100}
   LaserEnd_Ext()
   LIN {X 8.964, Y -5.478, Z 56.100}
   LaserStart_Ext()
   LIN {X -3.618, Y -5.478, Z 56.100}
   LaserEnd_Ext()
   LIN {X -3.868, Y -6.478, Z 56.100}
   LaserStart_Ext()
   LIN {X 8.944, Y -6.478, Z 56.100}
   LaserEnd_Ext()
   LIN {X 8.924, Y -7.478, Z 56.100}
   LaserStart_Ext()
   LIN {X -4.141, Y -7.478, Z 56.100}
   LaserEnd_Ext()
   LIN {X -4.471, Y -8.478, Z 56.100}
   LaserStart_Ext()
   LIN {X 8.865, Y -8.478, Z 56.100}
   LaserEnd_Ext()
   LIN {X 8.795, Y -9.478, Z 56.100}
   LaserStart_Ext()
   LIN {X -4.797, Y -9.478, Z 56.100}
   LaserEnd_Ext()
   LIN {X -5.122, Y -10.478, Z 56.100}
   LaserStart_Ext()
   LIN {X 8.722, Y -10.478, Z 56.100}
   LaserEnd_Ext()
   LIN {X 8.648, Y -11.478, Z 56.100}
   LaserStart_Ext()
   LIN {X -5.470, Y -11.478, Z 56.100}
   LaserEnd_Ext()
   LIN {X -5.854, Y -12.478, Z 56.100}
   LaserStart_Ext()
   LIN {X 8.571, Y -12.478, Z 56.100}
   LaserEnd_Ext()
   LIN {X 8.461, Y -13.478, Z 56.100}
   LaserStart_Ext()
   LIN {X -6.239, Y -13.478, Z 56.100}
   LaserEnd_Ext()
   LIN {X -6.630, Y -14.478, Z 56.100}
   LaserStart_Ext()
   LIN {X 8.352, Y -14.478, Z 56.100}
   LaserEnd_Ext()
   LIN {X 8.242, Y -15.478, Z 56.100}
   LaserStart_Ext()
   LIN {X 1.971, Y -15.478, Z 56.100}
   LaserEnd_Ext()
   LIN {X -3.322, Y -15.478, Z 56.100}
   LaserStart_Ext()
   LIN {X -7.060, Y -15.478, Z 56.100}
   LaserEnd_Ext()
   LIN {X -7.502, Y -16.478, Z 56.100}
   LaserStart_Ext()
   LIN {X -4.665, Y -16.478, Z 56.100}
   LaserEnd_Ext()
   LIN {X 3.532, Y -16.478, Z 56.100}
   LaserStart_Ext()
   LIN {X 8.115, Y -16.478, Z 56.100}
   LaserEnd_Ext()
   LIN {X 7.972, Y -17.478, Z 56.100}
   LaserStart_Ext()
   LIN {X 4.170, Y -17.478, Z 56.100}
   LaserEnd_Ext()
   LIN {X -5.641, Y -17.478, Z 56.100}
   LaserStart_Ext()
   LIN {X -7.920, Y -17.478, Z 56.100}
   LaserEnd_Ext()
   LIN {X -8.184, Y -18.478, Z 56.100}
   LaserStart_Ext()
   LIN {X -5.988, Y -18.478, Z 56.100}
   LaserEnd_Ext()
   LIN {X 4.778, Y -18.478, Z 56.100}
   LaserStart_Ext()
   LIN {X 7.831, Y -18.478, Z 56.100}
   LaserEnd_Ext()
   LIN {X 7.679, Y -19.478, Z 56.100}
   LaserStart_Ext()
   LIN {X 5.147, Y -19.478, Z 56.100}
   LaserEnd_Ext()
   LIN {X -6.324, Y -19.478, Z 56.100}
   LaserStart_Ext()
   LIN {X -8.452, Y -19.478, Z 56.100}
   LaserEnd_Ext()
   LIN {X -8.598, Y -20.478, Z 56.100}
   LaserStart_Ext()
   LIN {X -6.651, Y -20.478, Z 56.100}
   LaserEnd_Ext()
   LIN {X 5.209, Y -20.478, Z 56.100}
   LaserStart_Ext()
   LIN {X 7.511, Y -20.478, Z 56.100}
   LaserEnd_Ext()
   LIN {X 7.340, Y -21.478, Z 56.100}
   LaserStart_Ext()
   LIN {X 5.271, Y -21.478, Z 56.100}
   LaserEnd_Ext()
   LIN {X -6.542, Y -21.478, Z 56.100}
   LaserStart_Ext()
   LIN {X -8.476, Y -21.478, Z 56.100}
   LaserEnd_Ext()
   LIN {X -8.353, Y -22.478, Z 56.100}
   LaserStart_Ext()
   LIN {X -6.363, Y -22.478, Z 56.100}
   LaserEnd_Ext()
   LIN {X 4.968, Y -22.478, Z 56.100}
   LaserStart_Ext()
   LIN {X 7.073, Y -22.478, Z 56.100}
   LaserEnd_Ext()
   LIN {X 6.651, Y -23.478, Z 56.100}
   LaserStart_Ext()
   LIN {X 4.542, Y -23.478, Z 56.100}
   LaserEnd_Ext()
   LIN {X -5.997, Y -23.478, Z 56.100}
   LaserStart_Ext()
   LIN {X -8.209, Y -23.478, Z 56.100}
   LaserEnd_Ext()
   LIN {X -7.603, Y -24.478, Z 56.100}
   LaserStart_Ext()
   LIN {X -5.306, Y -24.478, Z 56.100}
   LaserEnd_Ext()
   LIN {X 4.041, Y -24.478, Z 56.100}
   LaserStart_Ext()
   LIN {X 6.239, Y -24.478, Z 56.100}
   LaserEnd_Ext()
   LIN {X 5.702, Y -25.478, Z 56.100}
   LaserStart_Ext()
   LIN {X 2.907, Y -25.478, Z 56.100}
   LaserEnd_Ext()
   LIN {X -4.338, Y -25.478, Z 56.100}
   LaserStart_Ext()
   LIN {X -7.001, Y -25.478, Z 56.100}
   LaserEnd_Ext()
   LIN {X -6.284, Y -26.478, Z 56.100}
   LaserStart_Ext()
   LIN {X -2.631, Y -26.478, Z 56.100}
   LaserEnd_Ext()
   LIN {X 0.828, Y -26.478, Z 56.100}
   LaserStart_Ext()
   LIN {X 4.698, Y -26.478, Z 56.100}
   LaserEnd_Ext()
   LIN {X 3.650, Y -27.478, Z 56.100}
   LaserStart_Ext()
   LIN {X -4.974, Y -27.478, Z 56.100}
   LaserEnd_Ext()
   LIN {X -0.694, Y -28.478, Z 56.100}
   LaserStart_Ext()
   LIN {X 1.061, Y -28.478, Z 56.100}
   LaserEnd_Ext()
   LIN {X -0.235, Y -25.728, Z 56.950}
   LaserStart_Ext()
   LIN {X -0.564, Y -25.687, Z 56.950} C_DIS
   LIN {X -2.265, Y -25.471, Z 56.950} C_DIS
   LIN {X -3.836, Y -24.517, Z 56.950} C_DIS
   LIN {X -4.030, Y -24.398, Z 56.950} C_DIS
   LIN {X -4.196, Y -24.157, Z 56.950} C_DIS
   LIN {X -5.219, Y -22.687, Z 56.950} C_DIS
   LIN {X -5.552, Y -20.867, Z 56.950} C_DIS
   LIN {X -5.593, Y -20.635, Z 56.950} C_DIS
   LIN {X -5.286, Y -19.719, Z 56.950} C_DIS
   LIN {X -4.664, Y -17.859, Z 56.950} C_DIS
   LIN {X -4.304, Y -17.525, Z 56.950} C_DIS
   LIN {X -3.144, Y -16.449, Z 56.950} C_DIS
   LIN {X -1.992, Y -16.072, Z 56.950} C_DIS
   LIN {X -1.056, Y -15.761, Z 56.950} C_DIS
   LIN {X 0.177, Y -15.899, Z 56.950} C_DIS
   LIN {X 1.075, Y -16.004, Z 56.950} C_DIS
   LIN {X 1.712, Y -16.397, Z 56.950} C_DIS
   LIN {X 2.886, Y -17.116, Z 56.950} C_DIS
   LIN {X 3.829, Y -18.657, Z 56.950} C_DIS
   LIN {X 4.211, Y -19.286, Z 56.950} C_DIS
   LIN {X 4.254, Y -19.967, Z 56.950} C_DIS
   LIN {X 4.354, Y -21.492, Z 56.950} C_DIS
   LIN {X 4.038, Y -22.243, Z 56.950} C_DIS
   LIN {X 3.409, Y -23.719, Z 56.950} C_DIS
   LIN {X 2.582, Y -24.451, Z 56.950} C_DIS
   LIN {X 1.852, Y -25.094, Z 56.950} C_DIS
   LIN {X 0.283, Y -25.570, Z 56.950} C_DIS
   LIN {X -0.235, Y -25.728, Z 56.950}
   LaserEnd_Ext()
   LIN {X 1.482, Y 40.353, Z 56.950}
   LaserStart_Ext()
   LIN {X 1.955, Y 39.217, Z 56.950} C_DIS
   LIN {X 2.449, Y 37.961, Z 56.950} C_DIS
   LIN {X 2.839, Y 36.968, Z 56.950} C_DIS
   LIN {X 3.109, Y 36.228, Z 56.950} C_DIS
   LIN {X 3.923, Y 33.993, Z 56.950} C_DIS
   LIN {X 4.592, Y 31.976, Z 56.950} C_DIS
   LIN {X 4.826, Y 31.270, Z 56.950} C_DIS
   LIN {X 6.500, Y 25.403, Z 56.950} C_DIS
   LIN {X 6.682, Y 24.813, Z 56.950} C_DIS
   LIN {X 6.750, Y 24.545, Z 56.950} C_DIS
   LIN {X 9.165, Y 11.841, Z 56.950} C_DIS
   LIN {X 9.198, Y 11.627, Z 56.950} C_DIS
   LIN {X 9.874, Y 4.485, Z 56.950} C_DIS
   LIN {X 9.940, Y 3.350, Z 56.950} C_DIS
   LIN {X 9.965, Y 2.566, Z 56.950} C_DIS
   LIN {X 10.084, Y -1.086, Z 56.950} C_DIS
   LIN {X 10.061, Y -2.893, Z 56.950} C_DIS
   LIN {X 9.968, Y -7.599, Z 56.950} C_DIS
   LIN {X 9.767, Y -10.621, Z 56.950} C_DIS
   LIN {X 9.638, Y -12.376, Z 56.950} C_DIS
   LIN {X 9.340, Y -15.099, Z 56.950} C_DIS
   LIN {X 9.228, Y -16.160, Z 56.950} C_DIS
   LIN {X 9.158, Y -16.678, Z 56.950} C_DIS
   LIN {X 8.819, Y -19.093, Z 56.950} C_DIS
   LIN {X 8.312, Y -22.127, Z 56.950} C_DIS
   LIN {X 8.279, Y -22.312, Z 56.950} C_DIS
   LIN {X 8.161, Y -22.593, Z 56.950} C_DIS
   LIN {X 6.994, Y -25.536, Z 56.950} C_DIS
   LIN {X 5.160, Y -27.473, Z 56.950} C_DIS
   LIN {X 4.363, Y -28.234, Z 56.950} C_DIS
   LIN {X 2.119, Y -29.097, Z 56.950} C_DIS
   LIN {X 0.802, Y -29.632, Z 56.950} C_DIS
   LIN {X 0.222, Y -29.571, Z 56.950} C_DIS
   LIN {X -3.844, Y -29.165, Z 56.950} C_DIS
   LIN {X -4.082, Y -29.058, Z 56.950} C_DIS
   LIN {X -4.853, Y -28.712, Z 56.950} C_DIS
   LIN {X -6.694, Y -27.311, Z 56.950} C_DIS
   LIN {X -7.167, Y -26.953, Z 56.950} C_DIS
   LIN {X -7.337, Y -26.677, Z 56.950} C_DIS
   LIN {X -9.111, Y -23.747, Z 56.950} C_DIS
   LIN {X -9.524, Y -20.497, Z 56.950} C_DIS
   LIN {X -9.577, Y -20.066, Z 56.950} C_DIS
   LIN {X -9.490, Y -19.743, Z 56.950} C_DIS
   LIN {X -8.768, Y -17.000, Z 56.950} C_DIS
   LIN {X -7.617, Y -14.374, Z 56.950} C_DIS
   LIN {X -7.541, Y -14.184, Z 56.950} C_DIS
   LIN {X -6.213, Y -10.729, Z 56.950} C_DIS
   LIN {X -5.186, Y -7.569, Z 56.950} C_DIS
   LIN {X -5.024, Y -7.061, Z 56.950} C_DIS
   LIN {X -4.754, Y -5.957, Z 56.950} C_DIS
   LIN {X -3.510, Y -0.970, Z 56.950} C_DIS
   LIN {X -3.322, Y 0.022, Z 56.950} C_DIS
   LIN {X -2.497, Y 5.442, Z 56.950} C_DIS
   LIN {X -2.284, Y 8.260, Z 56.950} C_DIS
   LIN {X -2.044, Y 13.313, Z 56.950} C_DIS
   LIN {X -2.445, Y 18.761, Z 56.950} C_DIS
   LIN {X -2.759, Y 23.765, Z 56.950} C_DIS
   LIN {X -3.694, Y 28.905, Z 56.950} C_DIS
   LIN {X -3.773, Y 29.347, Z 56.950} C_DIS
   LIN {X -3.818, Y 29.536, Z 56.950} C_DIS
   LIN {X -3.851, Y 29.672, Z 56.950} C_DIS
   LIN {X -4.045, Y 30.470, Z 56.950} C_DIS
   LIN {X -4.452, Y 32.149, Z 56.950} C_DIS
   LIN {X -4.682, Y 32.976, Z 56.950} C_DIS
   LIN {X -5.092, Y 34.432, Z 56.950} C_DIS
   LIN {X -5.759, Y 36.540, Z 56.950} C_DIS
   LIN {X -5.807, Y 36.693, Z 56.950} C_DIS
   LIN {X -6.330, Y 38.205, Z 56.950} C_DIS
   LIN {X -6.624, Y 39.021, Z 56.950} C_DIS
   LIN {X -6.755, Y 39.381, Z 56.950} C_DIS
   LIN {X -6.874, Y 40.009, Z 56.950} C_DIS
   LIN {X -7.022, Y 40.804, Z 56.950} C_DIS
   LIN {X -6.902, Y 41.446, Z 56.950} C_DIS
   LIN {X -6.747, Y 42.256, Z 56.950} C_DIS
   LIN {X -6.254, Y 43.012, Z 56.950} C_DIS
   LIN {X -5.911, Y 43.555, Z 56.950} C_DIS
   LIN {X -3.615, Y 44.659, Z 56.950} C_DIS
   LIN {X -3.409, Y 44.757, Z 56.950} C_DIS
   LIN {X -1.679, Y 44.529, Z 56.950} C_DIS
   LIN {X -0.340, Y 43.672, Z 56.950} C_DIS
   LIN {X -0.213, Y 43.591, Z 56.950} C_DIS
   LIN {X -0.129, Y 43.466, Z 56.950} C_DIS
   LIN {X 0.617, Y 42.375, Z 56.950} C_DIS
   LIN {X 1.062, Y 41.352, Z 56.950} C_DIS
   LIN {X 1.208, Y 41.014, Z 56.950} C_DIS
   LIN {X 1.482, Y 40.353, Z 56.950}
   LaserEnd_Ext()
   LIN {X -8.280, Y -19.074, Z 56.950}
   LaserStart_Ext()
   LIN {X -8.280, Y -22.356, Z 56.950}
   LaserEnd_Ext()
   LIN {X -7.280, Y -24.840, Z 56.950}
   LaserStart_Ext()
   LIN {X -7.280, Y -16.096, Z 56.950}
   LaserEnd_Ext()
   LIN {X -6.280, Y -13.690, Z 56.950}
   LaserStart_Ext()
   LIN {X -6.280, Y -19.537, Z 56.950}
   LaserEnd_Ext()
   LIN {X -6.280, Y -22.443, Z 56.950}
   LaserStart_Ext()
   LIN {X -6.280, Y -26.370, Z 56.950}
   LaserEnd_Ext()
   LIN {X -5.280, Y -27.131, Z 56.950}
   LaserStart_Ext()
   LIN {X -5.280, Y -24.351, Z 56.950}
   LaserEnd_Ext()
   LIN {X -5.280, Y -17.067, Z 56.950}
   LaserStart_Ext()
   LIN {X -5.280, Y -11.088, Z 56.950}
   LaserEnd_Ext()
   LIN {X -5.280, Y 38.228, Z 56.950}
   LaserStart_Ext()
   LIN {X -5.280, Y 42.682, Z 56.950}
   LaserEnd_Ext()
   LIN {X -4.280, Y 43.230, Z 56.950}
   LaserStart_Ext()
   LIN {X -4.280, Y 35.179, Z 56.950}
   LaserEnd_Ext()
   LIN {X -4.280, Y -8.016, Z 56.950}
   LaserStart_Ext()
   LIN {X -4.280, Y -16.138, Z 56.950}
   LaserEnd_Ext()
   LIN {X -4.280, Y -25.417, Z 56.950}
   LaserStart_Ext()
   LIN {X -4.280, Y -27.873, Z 56.950}
   LaserEnd_Ext()
   LIN {X -3.280, Y -28.217, Z 56.950}
   LaserStart_Ext()
   LIN {X -3.280, Y -26.025, Z 56.950}
   LaserEnd_Ext()
   LIN {X -3.280, Y -15.441, Z 56.950}
   LaserStart_Ext()
   LIN {X -3.280, Y -4.180, Z 56.950}
   LaserEnd_Ext()
   LIN {X -3.280, Y 31.558, Z 56.950}
   LaserStart_Ext()
   LIN {X -3.280, Y 43.711, Z 56.950}
   LaserEnd_Ext()
   LIN {X -2.280, Y 43.599, Z 56.950}
   LaserStart_Ext()
   LIN {X -2.280, Y 26.718, Z 56.950}
   LaserEnd_Ext()
   LIN {X -2.280, Y 0.225, Z 56.950}
   LaserStart_Ext()
   LIN {X -2.280, Y -15.114, Z 56.950}
   LaserEnd_Ext()
   LIN {X -2.280, Y -26.477, Z 56.950}
   LaserStart_Ext()
   LIN {X -2.280, Y -28.316, Z 56.950}
   LaserEnd_Ext()
   LIN {X -1.280, Y -28.416, Z 56.950}
   LaserStart_Ext()
   LIN {X -1.280, Y -26.604, Z 56.950}
   LaserEnd_Ext()
   LIN {X -1.280, Y -14.787, Z 56.950}
   LaserStart_Ext()
   LIN {X -1.280, Y 8.315, Z 56.950}
   LaserEnd_Ext()
   LIN {X -1.280, Y 16.554, Z 56.950}
   LaserStart_Ext()
   LIN {X -1.280, Y 43.086, Z 56.950}
   LaserEnd_Ext()
   LIN {X -0.280, Y 41.915, Z 56.950}
   LaserStart_Ext()
   LIN {X -0.280, Y -14.842, Z 56.950}
   LaserEnd_Ext()
   LIN {X -0.280, Y -26.726, Z 56.950}
   LaserStart_Ext()
   LIN {X -0.280, Y -28.516, Z 56.950}
   LaserEnd_Ext()
   LIN {X 0.720, Y -28.586, Z 56.950}
   LaserStart_Ext()
   LIN {X 0.720, Y -26.482, Z 56.950}
   LaserEnd_Ext()
   LIN {X 0.720, Y -14.956, Z 56.950}
   LaserStart_Ext()
   LIN {X 0.720, Y 39.581, Z 56.950}
   LaserEnd_Ext()
   LIN {X 1.720, Y 37.081, Z 56.950}
   LaserStart_Ext()
   LIN {X 1.720, Y -15.227, Z 56.950}
   LaserEnd_Ext()
   LIN {X 1.720, Y -26.179, Z 56.950}
   LaserStart_Ext()
   LIN {X 1.720, Y -28.180, Z 56.950}
   LaserEnd_Ext()
   LIN {X 2.720, Y -27.794, Z 56.950}
   LaserStart_Ext()
   LIN {X 2.720, Y -25.662, Z 56.950}
   LaserEnd_Ext()
   LIN {X 2.720, Y -15.842, Z 56.950}
   LaserStart_Ext()
   LIN {X 2.720, Y 34.373, Z 56.950}
   LaserEnd_Ext()
   LIN {X 3.720, Y 31.428, Z 56.950}
   LaserStart_Ext()
   LIN {X 3.720, Y -16.566, Z 56.950}
   LaserEnd_Ext()
   LIN {X 3.720, Y -24.779, Z 56.950}
   LaserStart_Ext()
   LIN {X 3.720, Y -27.409, Z 56.950}
   LaserEnd_Ext()
   LIN {X 4.720, Y -26.483, Z 56.950}
   LaserStart_Ext()
   LIN {X 4.720, Y -23.194, Z 56.950}
   LaserEnd_Ext()
   LIN {X 4.720, Y -18.197, Z 56.950}
   LaserStart_Ext()
   LIN {X 4.720, Y 27.997, Z 56.950}
   LaserEnd_Ext()
   LIN {X 5.720, Y 24.536, Z 56.950}
   LaserStart_Ext()
   LIN {X 5.720, Y -25.427, Z 56.950}
   LaserEnd_Ext()
   LIN {X 6.720, Y -23.514, Z 56.950}
   LaserStart_Ext()
   LIN {X 6.720, Y 19.349, Z 56.950}
   LaserEnd_Ext()
   LIN {X 7.720, Y 14.088, Z 56.950}
   LaserStart_Ext()
   LIN {X 7.720, Y -19.600, Z 56.950}
   LaserEnd_Ext()
   LIN {X 8.720, Y -11.221, Z 56.950}
   LaserStart_Ext()
   LIN {X 8.720, Y 6.061, Z 56.950}
   LaserEnd_Ext()
   LIN {X 1.142, Y -15.948, Z 57.800}
   LaserStart_Ext()
   LIN {X 1.783, Y -16.338, Z 57.800} C_DIS
   LIN {X 2.955, Y -17.056, Z 57.800} C_DIS
   LIN {X 3.729, Y -18.319, Z 57.800} C_DIS
   LIN {X 4.286, Y -19.223, Z 57.800} C_DIS
   LIN {X 4.346, Y -20.089, Z 57.800} C_DIS
   LIN {X 4.434, Y -21.428, Z 57.800} C_DIS
   LIN {X 3.778, Y -22.989, Z 57.800} C_DIS
   LIN {X 3.491, Y -23.663, Z 57.800} C_DIS
   LIN {X 2.228, Y -24.780, Z 57.800} C_DIS
   LIN {X 1.937, Y -25.039, Z 57.800} C_DIS
   LIN {X 1.699, Y -25.113, Z 57.800} C_DIS
   LIN {X -0.145, Y -25.675, Z 57.800} C_DIS
   LIN {X -1.709, Y -25.483, Z 57.800} C_DIS
   LIN {X -2.176, Y -25.424, Z 57.800} C_DIS
   LIN {X -2.735, Y -25.084, Z 57.800} C_DIS
   LIN {X -3.943, Y -24.354, Z 57.800} C_DIS
   LIN {X -4.633, Y -23.369, Z 57.800} C_DIS
   LIN {X -5.136, Y -22.646, Z 57.800} C_DIS
   LIN {X -5.290, Y -21.802, Z 57.800} C_DIS
   LIN {X -5.516, Y -20.595, Z 57.800} C_DIS
   LIN {X -5.199, Y -19.630, Z 57.800} C_DIS
   LIN {X -4.592, Y -17.817, Z 57.800} C_DIS
   LIN {X -3.141, Y -16.465, Z 57.800} C_DIS
   LIN {X -2.951, Y -16.361, Z 57.800} C_DIS
   LIN {X -0.995, Y -15.711, Z 57.800} C_DIS
   LIN {X 0.542, Y -15.884, Z 57.800} C_DIS
   LIN {X 1.142, Y -15.948, Z 57.800}
   LaserEnd_Ext()
   LIN {X 4.311, Y -28.226, Z 57.800}
   LaserStart_Ext()
   LIN {X 1.073, Y -29.542, Z 57.800} C_DIS
   LIN {X -0.720, Y -29.353, Z 57.800} C_DIS
   LIN {X -3.954, Y -29.031, Z 57.800} C_DIS
   LIN {X -4.756, Y -28.671, Z 57.800} C_DIS
   LIN {X -4.858, Y -28.594, Z 57.800} C_DIS
   LIN {X -7.075, Y -26.916, Z 57.800} C_DIS
   LIN {X -7.995, Y -25.419, Z 57.800} C_DIS
   LIN {X -9.026, Y -23.715, Z 57.800} C_DIS
   LIN {X -9.325, Y -21.363, Z 57.800} C_DIS
   LIN {X -9.500, Y -20.035, Z 57.800} C_DIS
   LIN {X -9.184, Y -18.812, Z 57.800} C_DIS
   LIN {X -8.699, Y -16.967, Z 57.800} C_DIS
   LIN {X -8.075, Y -15.544, Z 57.800} C_DIS
   LIN {X -7.522, Y -14.265, Z 57.800} C_DIS
   LIN {X -6.666, Y -12.012, Z 57.800} C_DIS
   LIN {X -6.160, Y -10.693, Z 57.800} C_DIS
   LIN {X -5.768, Y -9.487, Z 57.800} C_DIS
   LIN {X -4.978, Y -7.022, Z 57.800} C_DIS
   LIN {X -3.667, Y -1.659, Z 57.800} C_DIS
   LIN {X -3.438, Y -0.738, Z 57.800} C_DIS
   LIN {X -3.403, Y -0.555, Z 57.800} C_DIS
   LIN {X -2.470, Y 5.570, Z 57.800} C_DIS
   LIN {X -2.333, Y 7.384, Z 57.800} C_DIS
   LIN {X -2.046, Y 13.443, Z 57.800} C_DIS
   LIN {X -2.526, Y 19.975, Z 57.800} C_DIS
   LIN {X -2.753, Y 23.582, Z 57.800} C_DIS
   LIN {X -3.427, Y 27.287, Z 57.800} C_DIS
   LIN {X -3.761, Y 29.165, Z 57.800} C_DIS
   LIN {X -3.954, Y 29.969, Z 57.800} C_DIS
   LIN {X -4.095, Y 30.547, Z 57.800} C_DIS
   LIN {X -4.466, Y 32.073, Z 57.800} C_DIS
   LIN {X -4.953, Y 33.794, Z 57.800} C_DIS
   LIN {X -5.144, Y 34.473, Z 57.800} C_DIS
   LIN {X -5.277, Y 34.895, Z 57.800} C_DIS
   LIN {X -5.863, Y 36.732, Z 57.800} C_DIS
   LIN {X -6.325, Y 38.057, Z 57.800} C_DIS
   LIN {X -6.390, Y 38.243, Z 57.800} C_DIS
   LIN {X -6.485, Y 38.500, Z 57.800} C_DIS
   LIN {X -6.818, Y 39.418, Z 57.800} C_DIS
   LIN {X -6.958, Y 40.157, Z 57.800} C_DIS
   LIN {X -7.088, Y 40.843, Z 57.800} C_DIS
   LIN {X -6.935, Y 41.629, Z 57.800} C_DIS
   LIN {X -6.801, Y 42.333, Z 57.800} C_DIS
   LIN {X -6.410, Y 42.932, Z 57.800} C_DIS
   LIN {X -5.923, Y 43.656, Z 57.800} C_DIS
   LIN {X -5.001, Y 44.080, Z 57.800} C_DIS
   LIN {X -3.485, Y 44.802, Z 57.800} C_DIS
   LIN {X -2.078, Y 44.620, Z 57.800} C_DIS
   LIN {X -1.754, Y 44.578, Z 57.800} C_DIS
   LIN {X -1.445, Y 44.380, Z 57.800} C_DIS
   LIN {X -0.286, Y 43.643, Z 57.800} C_DIS
   LIN {X 0.389, Y 42.661, Z 57.800} C_DIS
   LIN {X 0.547, Y 42.430, Z 57.800} C_DIS
   LIN {X 0.684, Y 42.113, Z 57.800} C_DIS
   LIN {X 1.170, Y 41.001, Z 57.800} C_DIS
   LIN {X 1.659, Y 39.833, Z 57.800} C_DIS
   LIN {X 1.914, Y 39.222, Z 57.800} C_DIS
   LIN {X 2.265, Y 38.329, Z 57.800} C_DIS
   LIN {X 2.830, Y 36.901, Z 57.800} C_DIS
   LIN {X 3.863, Y 34.068, Z 57.800} C_DIS
   LIN {X 3.982, Y 33.739, Z 57.800} C_DIS
   LIN {X 4.026, Y 33.608, Z 57.800} C_DIS
   LIN {X 4.619, Y 31.822, Z 57.800} C_DIS
   LIN {X 5.798, Y 27.690, Z 57.800} C_DIS
   LIN {X 6.578, Y 25.151, Z 57.800} C_DIS
   LIN {X 6.874, Y 23.997, Z 57.800} C_DIS
   LIN {X 9.052, Y 12.541, Z 57.800} C_DIS
   LIN {X 9.286, Y 10.984, Z 57.800} C_DIS
   LIN {X 9.884, Y 4.670, Z 57.800} C_DIS
   LIN {X 9.992, Y 2.816, Z 57.800} C_DIS
   LIN {X 10.033, Y 1.533, Z 57.800} C_DIS
   LIN {X 10.116, Y -1.009, Z 57.800} C_DIS
   LIN {X 10.064, Y -5.042, Z 57.800} C_DIS
   LIN {X 10.015, Y -7.522, Z 57.800} C_DIS
   LIN {X 9.705, Y -12.183, Z 57.800} C_DIS
   LIN {X 9.696, Y -12.300, Z 57.800} C_DIS
   LIN {X 9.677, Y -12.483, Z 57.800} C_DIS
   LIN {X 9.296, Y -16.085, Z 57.800} C_DIS
   LIN {X 9.058, Y -17.844, Z 57.800} C_DIS
   LIN {X 8.893, Y -19.019, Z 57.800} C_DIS
   LIN {X 8.609, Y -20.721, Z 57.800} C_DIS
   LIN {X 8.361, Y -22.239, Z 57.800} C_DIS
   LIN {X 8.041, Y -23.145, Z 57.800} C_DIS
   LIN {X 7.185, Y -25.303, Z 57.800} C_DIS
   LIN {X 4.828, Y -27.793, Z 57.800} C_DIS
   LIN {X 4.537, Y -28.119, Z 57.800} C_DIS
   LIN {X 4.311, Y -28.226, Z 57.800}
   LaserEnd_Ext()
   LIN {X 1.325, Y -28.360, Z 57.800}
   LaserStart_Ext()
   LIN {X -0.604, Y -28.360, Z 57.800}
   LaserEnd_Ext()
   LIN {X -4.832, Y -27.360, Z 57.800}
   LaserStart_Ext()
   LIN {X 3.785, Y -27.360, Z 57.800}
   LaserEnd_Ext()
   LIN {X 4.807, Y -26.360, Z 57.800}
   LaserStart_Ext()
   LIN {X 1.037, Y -26.360, Z 57.800}
   LaserEnd_Ext()
   LIN {X -2.524, Y -26.360, Z 57.800}
   LaserStart_Ext()
   LIN {X -6.153, Y -26.360, Z 57.800}
   LaserEnd_Ext()
   LIN {X -6.857, Y -25.360, Z 57.800}
   LaserStart_Ext()
   LIN {X -4.212, Y -25.360, Z 57.800}
   LaserEnd_Ext()
   LIN {X 3.082, Y -25.360, Z 57.800}
   LaserStart_Ext()
   LIN {X 5.754, Y -25.360, Z 57.800}
   LaserEnd_Ext()
   LIN {X 6.483, Y -24.360, Z 57.800}
   LaserStart_Ext()
   LIN {X 4.207, Y -24.360, Z 57.800}
   LaserEnd_Ext()
   LIN {X -5.160, Y -24.360, Z 57.800}
   LaserStart_Ext()
   LIN {X -7.467, Y -24.360, Z 57.800}
   LaserEnd_Ext()
   LIN {X -8.063, Y -23.360, Z 57.800}
   LaserStart_Ext()
   LIN {X -5.858, Y -23.360, Z 57.800}
   LaserEnd_Ext()
   LIN {X 4.707, Y -23.360, Z 57.800}
   LaserStart_Ext()
   LIN {X 6.880, Y -23.360, Z 57.800}
   LaserEnd_Ext()
   LIN {X 7.258, Y -22.360, Z 57.800}
   LaserStart_Ext()
   LIN {X 5.127, Y -22.360, Z 57.800}
   LaserEnd_Ext()
   LIN {X -6.205, Y -22.360, Z 57.800}
   LaserStart_Ext()
   LIN {X -8.190, Y -22.360, Z 57.800}
   LaserEnd_Ext()
   LIN {X -8.317, Y -21.360, Z 57.800}
   LaserStart_Ext()
   LIN {X -6.390, Y -21.360, Z 57.800}
   LaserEnd_Ext()
   LIN {X 5.432, Y -21.360, Z 57.800}
   LaserStart_Ext()
   LIN {X 7.491, Y -21.360, Z 57.800}
   LaserEnd_Ext()
   LIN {X 7.655, Y -20.360, Z 57.800}
   LaserStart_Ext()
   LIN {X 5.366, Y -20.360, Z 57.800}
   LaserEnd_Ext()
   LIN {X -6.487, Y -20.360, Z 57.800}
   LaserStart_Ext()
   LIN {X -8.449, Y -20.360, Z 57.800}
   LaserEnd_Ext()
   LIN {X -8.293, Y -19.360, Z 57.800}
   LaserStart_Ext()
   LIN {X -6.163, Y -19.360, Z 57.800}
   LaserEnd_Ext()
   LIN {X 5.298, Y -19.360, Z 57.800}
   LaserStart_Ext()
   LIN {X 7.822, Y -19.360, Z 57.800}
   LaserEnd_Ext()
   LIN {X 7.976, Y -18.360, Z 57.800}
   LaserStart_Ext()
   LIN {X 4.929, Y -18.360, Z 57.800}
   LaserEnd_Ext()
   LIN {X -5.828, Y -18.360, Z 57.800}
   LaserStart_Ext()
   LIN {X -8.032, Y -18.360, Z 57.800}
   LaserEnd_Ext()
   LIN {X -7.768, Y -17.360, Z 57.800}
   LaserStart_Ext()
   LIN {X -5.480, Y -17.360, Z 57.800}
   LaserEnd_Ext()
   LIN {X 4.314, Y -17.360, Z 57.800}
   LaserStart_Ext()
   LIN {X 8.115, Y -17.360, Z 57.800}
   LaserEnd_Ext()
   LIN {X 8.249, Y -16.360, Z 57.800}
   LaserStart_Ext()
   LIN {X 3.672, Y -16.360, Z 57.800}
   LaserEnd_Ext()
   LIN {X -4.496, Y -16.360, Z 57.800}
   LaserStart_Ext()
   LIN {X -7.341, Y -16.360, Z 57.800}
   LaserEnd_Ext()
   LIN {X -6.906, Y -15.360, Z 57.800}
   LaserStart_Ext()
   LIN {X -3.109, Y -15.360, Z 57.800}
   LaserEnd_Ext()
   LIN {X 2.099, Y -15.360, Z 57.800}
   LaserStart_Ext()
   LIN {X 8.367, Y -15.360, Z 57.800}
   LaserEnd_Ext()
   LIN {X 8.472, Y -14.360, Z 57.800}
   LaserStart_Ext()
   LIN {X -6.488, Y -14.360, Z 57.800}
   LaserEnd_Ext()
   LIN {X -6.109, Y -13.360, Z 57.800}
   LaserStart_Ext()
   LIN {X 8.578, Y -13.360, Z 57.800}
   LaserEnd_Ext()
   LIN {X 8.684, Y -12.360, Z 57.800}
   LaserStart_Ext()
   LIN {X -5.729, Y -12.360, Z 57.800}
   LaserEnd_Ext()
   LIN {X -5.345, Y -11.360, Z 57.800}
   LaserStart_Ext()
   LIN {X 8.758, Y -11.360, Z 57.800}
   LaserEnd_Ext()
   LIN {X 8.824, Y -10.360, Z 57.800}
   LaserStart_Ext()
   LIN {X -5.000, Y -10.360, Z 57.800}
   LaserEnd_Ext()
   LIN {X -4.677, Y -9.360, Z 57.800}
   LaserStart_Ext()
   LIN {X 8.891, Y -9.360, Z 57.800}
   LaserEnd_Ext()
   LIN {X 8.957, Y -8.360, Z 57.800}
   LaserStart_Ext()
   LIN {X -4.357, Y -8.360, Z 57.800}
   LaserEnd_Ext()
   LIN {X -4.036, Y -7.360, Z 57.800}
   LaserStart_Ext()
   LIN {X 9.018, Y -7.360, Z 57.800}
   LaserEnd_Ext()
   LIN {X 9.038, Y -6.360, Z 57.800}
   LaserStart_Ext()
   LIN {X -3.787, Y -6.360, Z 57.800}
   LaserEnd_Ext()
   LIN {X -3.542, Y -5.360, Z 57.800}
   LaserStart_Ext()
   LIN {X 9.058, Y -5.360, Z 57.800}
   LaserEnd_Ext()
   LIN {X 9.073, Y -4.360, Z 57.800}
   LaserStart_Ext()
   LIN {X -3.298, Y -4.360, Z 57.800}
   LaserEnd_Ext()
   LIN {X -3.054, Y -3.360, Z 57.800}
   LaserStart_Ext()
   LIN {X 9.086, Y -3.360, Z 57.800}
   LaserEnd_Ext()
   LIN {X 9.098, Y -2.360, Z 57.800}
   LaserStart_Ext()
   LIN {X -2.809, Y -2.360, Z 57.800}
   LaserEnd_Ext()
   LIN {X -2.562, Y -1.360, Z 57.800}
   LaserStart_Ext()
   LIN {X 9.111, Y -1.360, Z 57.800}
   LaserEnd_Ext()
   LIN {X 9.094, Y -0.360, Z 57.800}
   LaserStart_Ext()
   LIN {X -2.362, Y -0.360, Z 57.800}
   LaserEnd_Ext()
   LIN {X -2.210, Y 0.640, Z 57.800}
   LaserStart_Ext()
   LIN {X 9.062, Y 0.640, Z 57.800}
   LaserEnd_Ext()
   LIN {X 9.029, Y 1.640, Z 57.800}
   LaserStart_Ext()
   LIN {X -2.057, Y 1.640, Z 57.800}
   LaserEnd_Ext()
   LIN {X -1.905, Y 2.640, Z 57.800}
   LaserStart_Ext()
   LIN {X 8.997, Y 2.640, Z 57.800}
   LaserEnd_Ext()
   LIN {X 8.942, Y 3.640, Z 57.800}
   LaserStart_Ext()
   LIN {X -1.753, Y 3.640, Z 57.800}
   LaserEnd_Ext()
   LIN {X -1.601, Y 4.640, Z 57.800}
   LaserStart_Ext()
   LIN {X 8.882, Y 4.640, Z 57.800}
   LaserEnd_Ext()
   LIN {X 8.787, Y 5.640, Z 57.800}
   LaserStart_Ext()
   LIN {X -1.462, Y 5.640, Z 57.800}
   LaserEnd_Ext()
   LIN {X -1.387, Y 6.640, Z 57.800}
   LaserStart_Ext()
   LIN {X 8.693, Y 6.640, Z 57.800}
   LaserEnd_Ext()
   LIN {X 8.598, Y 7.640, Z 57.800}
   LaserStart_Ext()
   LIN {X -1.320, Y 7.640, Z 57.800}
   LaserEnd_Ext()
   LIN {X -1.272, Y 8.640, Z 57.800}
   LaserStart_Ext()
   LIN {X 8.503, Y 8.640, Z 57.800}
   LaserEnd_Ext()
   LIN {X 8.409, Y 9.640, Z 57.800}
   LaserStart_Ext()
   LIN {X -1.225, Y 9.640, Z 57.800}
   LaserEnd_Ext()
   LIN {X -1.178, Y 10.640, Z 57.800}
   LaserStart_Ext()
   LIN {X 8.314, Y 10.640, Z 57.800}
   LaserEnd_Ext()
   LIN {X 8.176, Y 11.640, Z 57.800}
   LaserStart_Ext()
   LIN {X -1.130, Y 11.640, Z 57.800}
   LaserEnd_Ext()
   LIN {X -1.083, Y 12.640, Z 57.800}
   LaserStart_Ext()
   LIN {X 8.015, Y 12.640, Z 57.800}
   LaserEnd_Ext()
   LIN {X 7.825, Y 13.640, Z 57.800}
   LaserStart_Ext()
   LIN {X -1.058, Y 13.640, Z 57.800}
   LaserEnd_Ext()
   LIN {X -1.131, Y 14.640, Z 57.800}
   LaserStart_Ext()
   LIN {X 7.635, Y 14.640, Z 57.800}
   LaserEnd_Ext()
   LIN {X 7.445, Y 15.640, Z 57.800}
   LaserStart_Ext()
   LIN {X -1.205, Y 15.640, Z 57.800}
   LaserEnd_Ext()
   LIN {X -1.278, Y 16.640, Z 57.800}
   LaserStart_Ext()
   LIN {X 7.255, Y 16.640, Z 57.800}
   LaserEnd_Ext()
   LIN {X 7.064, Y 17.640, Z 57.800}
   LaserStart_Ext()
   LIN {X -1.352, Y 17.640, Z 57.800}
   LaserEnd_Ext()
   LIN {X -1.426, Y 18.640, Z 57.800}
   LaserStart_Ext()
   LIN {X 6.874, Y 18.640, Z 57.800}
   LaserEnd_Ext()
   LIN {X 6.684, Y 19.640, Z 57.800}
   LaserStart_Ext()
   LIN {X -1.499, Y 19.640, Z 57.800}
   LaserEnd_Ext()
   LIN {X -1.566, Y 20.640, Z 57.800}
   LaserStart_Ext()
   LIN {X 6.494, Y 20.640, Z 57.800}
   LaserEnd_Ext()
   LIN {X 6.304, Y 21.640, Z 57.800}
   LaserStart_Ext()
   LIN {X -1.629, Y 21.640, Z 57.800}
   LaserEnd_Ext()
   LIN {X -1.692, Y 22.640, Z 57.800}
   LaserStart_Ext()
   LIN {X 6.114, Y 22.640, Z 57.800}
   LaserEnd_Ext()
   LIN {X 5.924, Y 23.640, Z 57.800}
   LaserStart_Ext()
   LIN {X -1.755, Y 23.640, Z 57.800}
   LaserEnd_Ext()
   LIN {X -1.929, Y 24.640, Z 57.800}
   LaserStart_Ext()
   LIN {X 5.677, Y 24.640, Z 57.800}
   LaserEnd_Ext()
   LIN {X 5.382, Y 25.640, Z 57.800}
   LaserStart_Ext()
   LIN {X -2.111, Y 25.640, Z 57.800}
   LaserEnd_Ext()
   LIN {X -2.293, Y 26.640, Z 57.800}
   LaserStart_Ext()
   LIN {X 5.075, Y 26.640, Z 57.800}
   LaserEnd_Ext()
   LIN {X 4.773, Y 27.640, Z 57.800}
   LaserStart_Ext()
   LIN {X -2.474, Y 27.640, Z 57.800}
   LaserEnd_Ext()
   LIN {X -2.652, Y 28.640, Z 57.800}
   LaserStart_Ext()
   LIN {X 4.487, Y 28.640, Z 57.800}
   LaserEnd_Ext()
   LIN {X 4.202, Y 29.640, Z 57.800}
   LaserStart_Ext()
   LIN {X -2.847, Y 29.640, Z 57.800}
   LaserEnd_Ext()
   LIN {X -3.088, Y 30.640, Z 57.800}
   LaserStart_Ext()
   LIN {X 3.917, Y 30.640, Z 57.800}
   LaserEnd_Ext()
   LIN {X 3.626, Y 31.640, Z 57.800}
   LaserStart_Ext()
   LIN {X -3.332, Y 31.640, Z 57.800}
   LaserEnd_Ext()
   LIN {X -3.587, Y 32.640, Z 57.800}
   LaserStart_Ext()
   LIN {X 3.294, Y 32.640, Z 57.800}
   LaserEnd_Ext()
   LIN {X 2.954, Y 33.640, Z 57.800}
   LaserStart_Ext()
   LIN {X -3.870, Y 33.640, Z 57.800}
   LaserEnd_Ext()
   LIN {X -4.152, Y 34.640, Z 57.800}
   LaserStart_Ext()
   LIN {X 2.590, Y 34.640, Z 57.800}
   LaserEnd_Ext()
   LIN {X 2.225, Y 35.640, Z 57.800}
   LaserStart_Ext()
   LIN {X -4.465, Y 35.640, Z 57.800}
   LaserEnd_Ext()
   LIN {X -4.785, Y 36.640, Z 57.800}
   LaserStart_Ext()
   LIN {X 1.858, Y 36.640, Z 57.800}
   LaserEnd_Ext()
   LIN {X 1.462, Y 37.640, Z 57.800}
   LaserStart_Ext()
   LIN {X -5.121, Y 37.640, Z 57.800}
   LaserEnd_Ext()
   LIN {X -5.471, Y 38.640, Z 57.800}
   LaserStart_Ext()
   LIN {X 1.068, Y 38.640, Z 57.800}
   LaserEnd_Ext()
   LIN {X 0.656, Y 39.640, Z 57.800}
   LaserStart_Ext()
   LIN {X -5.835, Y 39.640, Z 57.800}
   LaserEnd_Ext()
   LIN {X -6.032, Y 40.640, Z 57.800}
   LaserStart_Ext()
   LIN {X 0.237, Y 40.640, Z 57.800}
   LaserEnd_Ext()
   LIN {X -0.200, Y 41.640, Z 57.800}
   LaserStart_Ext()
   LIN {X -5.915, Y 41.640, Z 57.800}
   LaserEnd_Ext()
   LIN {X -5.401, Y 42.640, Z 57.800}
   LaserStart_Ext()
   LIN {X -0.810, Y 42.640, Z 57.800}
   LaserEnd_Ext()
   LIN {X -2.294, Y 43.640, Z 57.800}
   LaserStart_Ext()
   LIN {X -3.599, Y 43.640, Z 57.800}
   LaserEnd_Ext()
   LIN {X -3.967, Y -17.259, Z 58.650}
   LaserStart_Ext()
   LIN {X -3.010, Y -16.359, Z 58.650} C_DIS
   LIN {X -1.184, Y -15.744, Z 58.650} C_DIS
   LIN {X -0.934, Y -15.661, Z 58.650} C_DIS
   LIN {X -0.738, Y -15.683, Z 58.650} C_DIS
   LIN {X 1.209, Y -15.893, Z 58.650} C_DIS
   LIN {X 2.813, Y -16.868, Z 58.650} C_DIS
   LIN {X 3.025, Y -16.996, Z 58.650} C_DIS
   LIN {X 3.197, Y -17.273, Z 58.650} C_DIS
   LIN {X 4.361, Y -19.160, Z 58.650} C_DIS
   LIN {X 4.503, Y -21.209, Z 58.650} C_DIS
   LIN {X 4.514, Y -21.365, Z 58.650} C_DIS
   LIN {X 3.572, Y -23.607, Z 58.650} C_DIS
   LIN {X 3.425, Y -23.738, Z 58.650} C_DIS
   LIN {X 2.025, Y -24.981, Z 58.650} C_DIS
   LIN {X 0.563, Y -25.434, Z 58.650} C_DIS
   LIN {X -0.056, Y -25.622, Z 58.650} C_DIS
   LIN {X -0.966, Y -25.511, Z 58.650} C_DIS
   LIN {X -2.087, Y -25.376, Z 58.650} C_DIS
   LIN {X -2.815, Y -24.940, Z 58.650} C_DIS
   LIN {X -3.857, Y -24.310, Z 58.650} C_DIS
   LIN {X -4.681, Y -23.134, Z 58.650} C_DIS
   LIN {X -5.053, Y -22.606, Z 58.650} C_DIS
   LIN {X -5.178, Y -21.951, Z 58.650} C_DIS
   LIN {X -5.438, Y -20.555, Z 58.650} C_DIS
   LIN {X -4.753, Y -18.467, Z 58.650} C_DIS
   LIN {X -4.521, Y -17.775, Z 58.650} C_DIS
   LIN {X -3.967, Y -17.259, Z 58.650}
   LaserEnd_Ext()
   LIN {X 1.146, Y 40.959, Z 58.650}
   LaserStart_Ext()
   LIN {X 1.488, Y 40.141, Z 58.650} C_DIS
   LIN {X 1.907, Y 39.143, Z 58.650} C_DIS
   LIN {X 2.504, Y 37.637, Z 58.650} C_DIS
   LIN {X 2.793, Y 36.907, Z 58.650} C_DIS
   LIN {X 3.073, Y 36.140, Z 58.650} C_DIS
   LIN {X 4.043, Y 33.486, Z 58.650} C_DIS
   LIN {X 4.412, Y 32.374, Z 58.650} C_DIS
   LIN {X 5.096, Y 29.978, Z 58.650} C_DIS
   LIN {X 6.474, Y 25.489, Z 58.650} C_DIS
   LIN {X 6.997, Y 23.450, Z 58.650} C_DIS
   LIN {X 8.938, Y 13.241, Z 58.650} C_DIS
   LIN {X 9.374, Y 10.341, Z 58.650} C_DIS
   LIN {X 9.894, Y 4.855, Z 58.650} C_DIS
   LIN {X 10.044, Y 2.281, Z 58.650} C_DIS
   LIN {X 10.101, Y 0.500, Z 58.650} C_DIS
   LIN {X 10.148, Y -0.932, Z 58.650} C_DIS
   LIN {X 10.068, Y -7.192, Z 58.650} C_DIS
   LIN {X 10.063, Y -7.446, Z 58.650} C_DIS
   LIN {X 10.028, Y -7.969, Z 58.650} C_DIS
   LIN {X 9.755, Y -12.224, Z 58.650} C_DIS
   LIN {X 9.638, Y -13.411, Z 58.650} C_DIS
   LIN {X 9.363, Y -16.010, Z 58.650} C_DIS
   LIN {X 8.977, Y -18.872, Z 58.650} C_DIS
   LIN {X 8.958, Y -19.007, Z 58.650} C_DIS
   LIN {X 8.443, Y -22.166, Z 58.650} C_DIS
   LIN {X 7.743, Y -24.145, Z 58.650} C_DIS
   LIN {X 7.377, Y -25.069, Z 58.650} C_DIS
   LIN {X 6.367, Y -26.135, Z 58.650} C_DIS
   LIN {X 4.709, Y -28.000, Z 58.650} C_DIS
   LIN {X 3.418, Y -28.609, Z 58.650} C_DIS
   LIN {X 1.344, Y -29.452, Z 58.650} C_DIS
   LIN {X -1.662, Y -29.136, Z 58.650} C_DIS
   LIN {X -4.063, Y -28.896, Z 58.650} C_DIS
   LIN {X -4.659, Y -28.629, Z 58.650} C_DIS
   LIN {X -5.605, Y -27.922, Z 58.650} C_DIS
   LIN {X -6.982, Y -26.880, Z 58.650} C_DIS
   LIN {X -8.652, Y -24.161, Z 58.650} C_DIS
   LIN {X -8.941, Y -23.684, Z 58.650} C_DIS
   LIN {X -9.025, Y -23.025, Z 58.650} C_DIS
   LIN {X -9.424, Y -20.004, Z 58.650} C_DIS
   LIN {X -8.706, Y -17.223, Z 58.650} C_DIS
   LIN {X -8.630, Y -16.935, Z 58.650} C_DIS
   LIN {X -8.533, Y -16.713, Z 58.650} C_DIS
   LIN {X -7.456, Y -14.224, Z 58.650} C_DIS
   LIN {X -6.324, Y -11.240, Z 58.650} C_DIS
   LIN {X -6.105, Y -10.654, Z 58.650} C_DIS
   LIN {X -5.898, Y -9.997, Z 58.650} C_DIS
   LIN {X -4.933, Y -6.983, Z 58.650} C_DIS
   LIN {X -3.860, Y -2.594, Z 58.650} C_DIS
   LIN {X -3.397, Y -0.652, Z 58.650} C_DIS
   LIN {X -2.932, Y 2.490, Z 58.650} C_DIS
   LIN {X -2.444, Y 5.698, Z 58.650} C_DIS
   LIN {X -2.383, Y 6.508, Z 58.650} C_DIS
   LIN {X -2.048, Y 13.572, Z 58.650} C_DIS
   LIN {X -2.608, Y 21.189, Z 58.650} C_DIS
   LIN {X -2.747, Y 23.400, Z 58.650} C_DIS
   LIN {X -3.160, Y 25.670, Z 58.650} C_DIS
   LIN {X -3.749, Y 28.983, Z 58.650} C_DIS
   LIN {X -4.089, Y 30.401, Z 58.650} C_DIS
   LIN {X -4.338, Y 31.421, Z 58.650} C_DIS
   LIN {X -4.451, Y 31.882, Z 58.650} C_DIS
   LIN {X -4.697, Y 32.753, Z 58.650} C_DIS
   LIN {X -5.195, Y 34.513, Z 58.650} C_DIS
   LIN {X -5.808, Y 36.420, Z 58.650} C_DIS
   LIN {X -5.920, Y 36.771, Z 58.650} C_DIS
   LIN {X -5.978, Y 36.937, Z 58.650} C_DIS
   LIN {X -6.450, Y 38.280, Z 58.650} C_DIS
   LIN {X -6.744, Y 39.083, Z 58.650} C_DIS
   LIN {X -6.881, Y 39.455, Z 58.650} C_DIS
   LIN {X -7.010, Y 40.126, Z 58.650} C_DIS
   LIN {X -7.154, Y 40.883, Z 58.650} C_DIS
   LIN {X -7.012, Y 41.614, Z 58.650} C_DIS
   LIN {X -6.854, Y 42.410, Z 58.650} C_DIS
   LIN {X -6.332, Y 43.165, Z 58.650} C_DIS
   LIN {X -5.934, Y 43.756, Z 58.650} C_DIS
   LIN {X -3.970, Y 44.660, Z 58.650} C_DIS
   LIN {X -3.560, Y 44.846, Z 58.650} C_DIS
   LIN {X -3.443, Y 44.831, Z 58.650} C_DIS
   LIN {X -1.829, Y 44.626, Z 58.650} C_DIS
   LIN {X -0.899, Y 44.038, Z 58.650} C_DIS
   LIN {X -0.359, Y 43.694, Z 58.650} C_DIS
   LIN {X -0.059, Y 43.259, Z 58.650} C_DIS
   LIN {X 0.477, Y 42.483, Z 58.650} C_DIS
   LIN {X 0.884, Y 41.559, Z 58.650} C_DIS
   LIN {X 1.146, Y 40.959, Z 58.650}
   LaserEnd_Ext()
   LIN {X 8.602, Y 7.888, Z 58.650}
   LaserStart_Ext()
   LIN {X 8.602, Y -13.698, Z 58.650}
   LaserEnd_Ext()
   LIN {X 7.602, Y -21.112, Z 58.650}
   LaserStart_Ext()
   LIN {X 7.602, Y 14.914, Z 58.650}
   LaserEnd_Ext()
   LIN {X 6.602, Y 20.175, Z 58.650}
   LaserStart_Ext()
   LIN {X 6.602, Y -24.310, Z 58.650}
   LaserEnd_Ext()
   LIN {X 5.602, Y -25.491, Z 58.650}
   LaserStart_Ext()
   LIN {X 5.602, Y 24.866, Z 58.650}
   LaserEnd_Ext()
   LIN {X 4.602, Y 28.180, Z 58.650}
   LaserStart_Ext()
   LIN {X 4.602, Y -17.646, Z 58.650}
   LaserEnd_Ext()
   LIN {X 4.602, Y -23.738, Z 58.650}
   LaserStart_Ext()
   LIN {X 4.602, Y -26.615, Z 58.650}
   LaserEnd_Ext()
   LIN {X 3.602, Y -27.416, Z 58.650}
   LaserStart_Ext()
   LIN {X 3.602, Y -24.918, Z 58.650}
   LaserEnd_Ext()
   LIN {X 3.602, Y -16.180, Z 58.650}
   LaserStart_Ext()
   LIN {X 3.602, Y 31.570, Z 58.650}
   LaserEnd_Ext()
   LIN {X 2.602, Y 34.515, Z 58.650}
   LaserStart_Ext()
   LIN {X 2.602, Y -15.569, Z 58.650}
   LaserEnd_Ext()
   LIN {X 2.602, Y -25.798, Z 58.650}
   LaserStart_Ext()
   LIN {X 2.602, Y -27.861, Z 58.650}
   LaserEnd_Ext()
   LIN {X 1.602, Y -28.267, Z 58.650}
   LaserStart_Ext()
   LIN {X 1.602, Y -26.159, Z 58.650}
   LaserEnd_Ext()
   LIN {X 1.602, Y -14.975, Z 58.650}
   LaserStart_Ext()
   LIN {X 1.602, Y 37.200, Z 58.650}
   LaserEnd_Ext()
   LIN {X 0.602, Y 39.668, Z 58.650}
   LaserStart_Ext()
   LIN {X 0.602, Y -14.822, Z 58.650}
   LaserEnd_Ext()
   LIN {X 0.602, Y -26.467, Z 58.650}
   LaserStart_Ext()
   LIN {X 0.602, Y -28.368, Z 58.650}
   LaserEnd_Ext()
   LIN {X -0.398, Y -28.263, Z 58.650}
   LaserStart_Ext()
   LIN {X -0.398, Y -26.588, Z 58.650}
   LaserEnd_Ext()
   LIN {X -0.398, Y -14.714, Z 58.650}
   LaserStart_Ext()
   LIN {X -0.398, Y 41.989, Z 58.650}
   LaserEnd_Ext()
   LIN {X -1.398, Y 43.170, Z 58.650}
   LaserStart_Ext()
   LIN {X -1.398, Y 18.371, Z 58.650}
   LaserEnd_Ext()
   LIN {X -1.398, Y 6.266, Z 58.650}
   LaserStart_Ext()
   LIN {X -1.398, Y -14.761, Z 58.650}
   LaserEnd_Ext()
   LIN {X -1.398, Y -26.466, Z 58.650}
   LaserStart_Ext()
   LIN {X -1.398, Y -28.158, Z 58.650}
   LaserEnd_Ext()
   LIN {X -2.398, Y -28.057, Z 58.650}
   LaserStart_Ext()
   LIN {X -2.398, Y -26.325, Z 58.650}
   LaserEnd_Ext()
   LIN {X -2.398, Y -15.098, Z 58.650}
   LaserStart_Ext()
   LIN {X -2.398, Y -0.731, Z 58.650}
   LaserEnd_Ext()
   LIN {X -2.398, Y 27.097, Z 58.650}
   LaserStart_Ext()
   LIN {X -2.398, Y 43.690, Z 58.650}
   LaserEnd_Ext()
   LIN {X -3.398, Y 43.818, Z 58.650}
   LaserStart_Ext()
   LIN {X -3.398, Y 31.787, Z 58.650}
   LaserEnd_Ext()
   LIN {X -3.398, Y -4.916, Z 58.650}
   LaserStart_Ext()
   LIN {X -3.398, Y -15.439, Z 58.650}
   LaserEnd_Ext()
   LIN {X -3.398, Y -25.756, Z 58.650}
   LaserStart_Ext()
   LIN {X -3.398, Y -27.957, Z 58.650}
   LaserEnd_Ext()
   LIN {X -4.398, Y -27.576, Z 58.650}
   LaserStart_Ext()
   LIN {X -4.398, Y -25.150, Z 58.650}
   LaserEnd_Ext()
   LIN {X -4.398, Y -16.292, Z 58.650}
